REGION Network 5: создаем лог
   #_w1 := "data".executeCreate AND NOT #DL.stateMem;   // rising edge of "data".executeCreate
   #DL.stateMem := "data".executeCreate;
   #DataLogCreate_Instance(REQ := #_w1,   // DataLogCreate
                           RECORDS := 3000,
                           "NAME" := "data"."name",
                           ID := "data".logID,
                           DATA := "data".myData,
                           DONE => "data".crateDone,
                           BUSY => "data".createBusy,
                           ERROR => "data".createError,
                           STATUS => "data".createStatus);
END_REGION

REGION Network 6: если ошибка
   RUNG wire#powerrail
      Contact( "data".createError )
      Move(in := "data".createStatus, out1 => "data".createStatusMem)
   END_RUNG
   // the same network as SCL:
   IF "data".createError THEN "data".createStatusMem := "data".createStatus; END_IF;
END_REGION

REGION Network 7: создана сессия
   RUNG wire#powerrail
      Contact( "data".crateDone )
      S_Coil( "data".dlogCreated )
   END_RUNG
   // the same network as SCL:
   IF "data".crateDone THEN "data".dlogCreated := TRUE; END_IF;
END_REGION

REGION Network 8: запись значений в бд
   RUNG wire#powerrail
      P_Contact(operand := "logW".executeWrite, bit := #DL.stateMem_2)
      Move(in := "T3V3W3_DB".Statistic.Count, out1 => "data".myData.number)
      Move(in := "T3V3W3_DB".LocalVar.SP_loaded, out1 => "data".myData.weight)
   END_RUNG
   // the same network as SCL:
   #_w1 := "logW".executeWrite AND NOT #DL.stateMem_2;   // rising edge of "logW".executeWrite
   #DL.stateMem_2 := "logW".executeWrite;
   IF #_w1 THEN
       "data".myData.number := "T3V3W3_DB".Statistic.Count;
       "data".myData.weight := "T3V3W3_DB".LocalVar.SP_loaded;
   END_IF;
END_REGION

REGION Network 9: запись на флеш
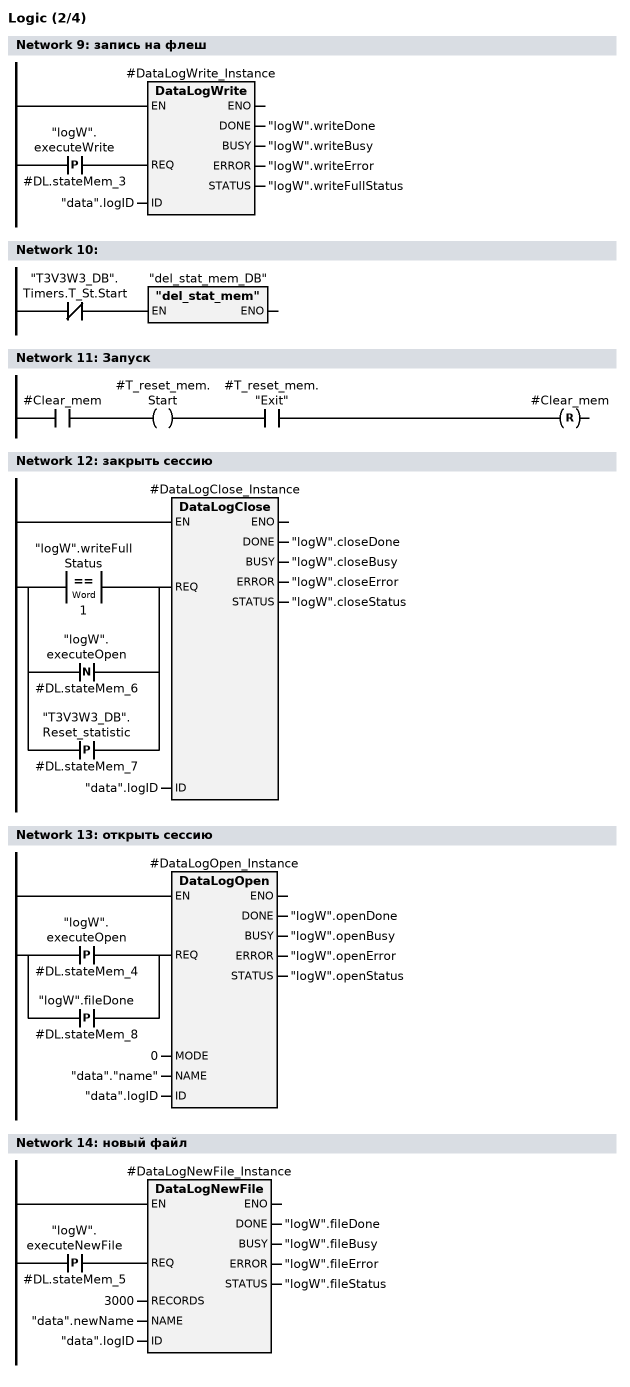
   #_w1 := "logW".executeWrite AND NOT #DL.stateMem_3;   // rising edge of "logW".executeWrite
   #DL.stateMem_3 := "logW".executeWrite;
   #DataLogWrite_Instance(REQ := #_w1,   // DataLogWrite
                          ID := "data".logID,
                          DONE => "logW".writeDone,
                          BUSY => "logW".writeBusy,
                          ERROR => "logW".writeError,
                          STATUS => "logW".writeFullStatus);
END_REGION

REGION Network 10
   RUNG wire#powerrail
      I_Contact( "T3V3W3_DB".Timers.T_St.Start )
      "del_stat_mem_DB"()
   END_RUNG
   // the same network as SCL:
   IF NOT "T3V3W3_DB".Timers.T_St.Start THEN
       "del_stat_mem_DB"();   // "del_stat_mem"
   END_IF;
END_REGION

REGION Network 11: Запуск
   RUNG wire#powerrail
      Contact( #Clear_mem )
      Coil( #T_reset_mem.Start )
      Contact( #T_reset_mem."Exit" )
      R_Coil( #Clear_mem )
   END_RUNG
   // the same network as SCL:
   #T_reset_mem.Start := #Clear_mem;
   IF #Clear_mem AND #T_reset_mem."Exit" THEN #Clear_mem := FALSE; END_IF;
END_REGION

REGION Network 12: закрыть сессию
   #_w1 := NOT "logW".executeOpen AND #DL.stateMem_6;   // falling edge of "logW".executeOpen
   #DL.stateMem_6 := "logW".executeOpen;
   #_w2 := "T3V3W3_DB".Reset_statistic AND NOT #DL.stateMem_7;   // rising edge of "T3V3W3_DB".Reset_statistic
   #DL.stateMem_7 := "T3V3W3_DB".Reset_statistic;
   #DataLogClose_Instance(REQ := ("logW".writeFullStatus = 1) OR #_w1 OR #_w2,   // DataLogClose
                          ID := "data".logID,
                          DONE => "logW".closeDone,
                          BUSY => "logW".closeBusy,
                          ERROR => "logW".closeError,
                          STATUS => "logW".closeStatus);
END_REGION

REGION Network 13: открыть сессию
   #_w1 := "logW".executeOpen AND NOT #DL.stateMem_4;   // rising edge of "logW".executeOpen
   #DL.stateMem_4 := "logW".executeOpen;
   #_w2 := "logW".fileDone AND NOT #DL.stateMem_8;   // rising edge of "logW".fileDone
   #DL.stateMem_8 := "logW".fileDone;
   #DataLogOpen_Instance(REQ := #_w1 OR #_w2,   // DataLogOpen
                         MODE := 0,
                         "NAME" := "data"."name",
                         ID := "data".logID,
                         DONE => "logW".openDone,
                         BUSY => "logW".openBusy,
                         ERROR => "logW".openError,
                         STATUS => "logW".openStatus);
END_REGION

REGION Network 14: новый файл
   #_w1 := "logW".executeNewFile AND NOT #DL.stateMem_5;   // rising edge of "logW".executeNewFile
   #DL.stateMem_5 := "logW".executeNewFile;
   #DataLogNewFile_Instance(REQ := #_w1,   // DataLogNewFile
                           RECORDS := 3000,
                           "NAME" := "data".newName,
                           ID := "data".logID,
                           DONE => "logW".fileDone,
                           BUSY => "logW".fileBusy,
                           ERROR => "logW".fileError,
                           STATUS => "logW".fileStatus);
END_REGION

REGION Network 16: Сброс команды на запись
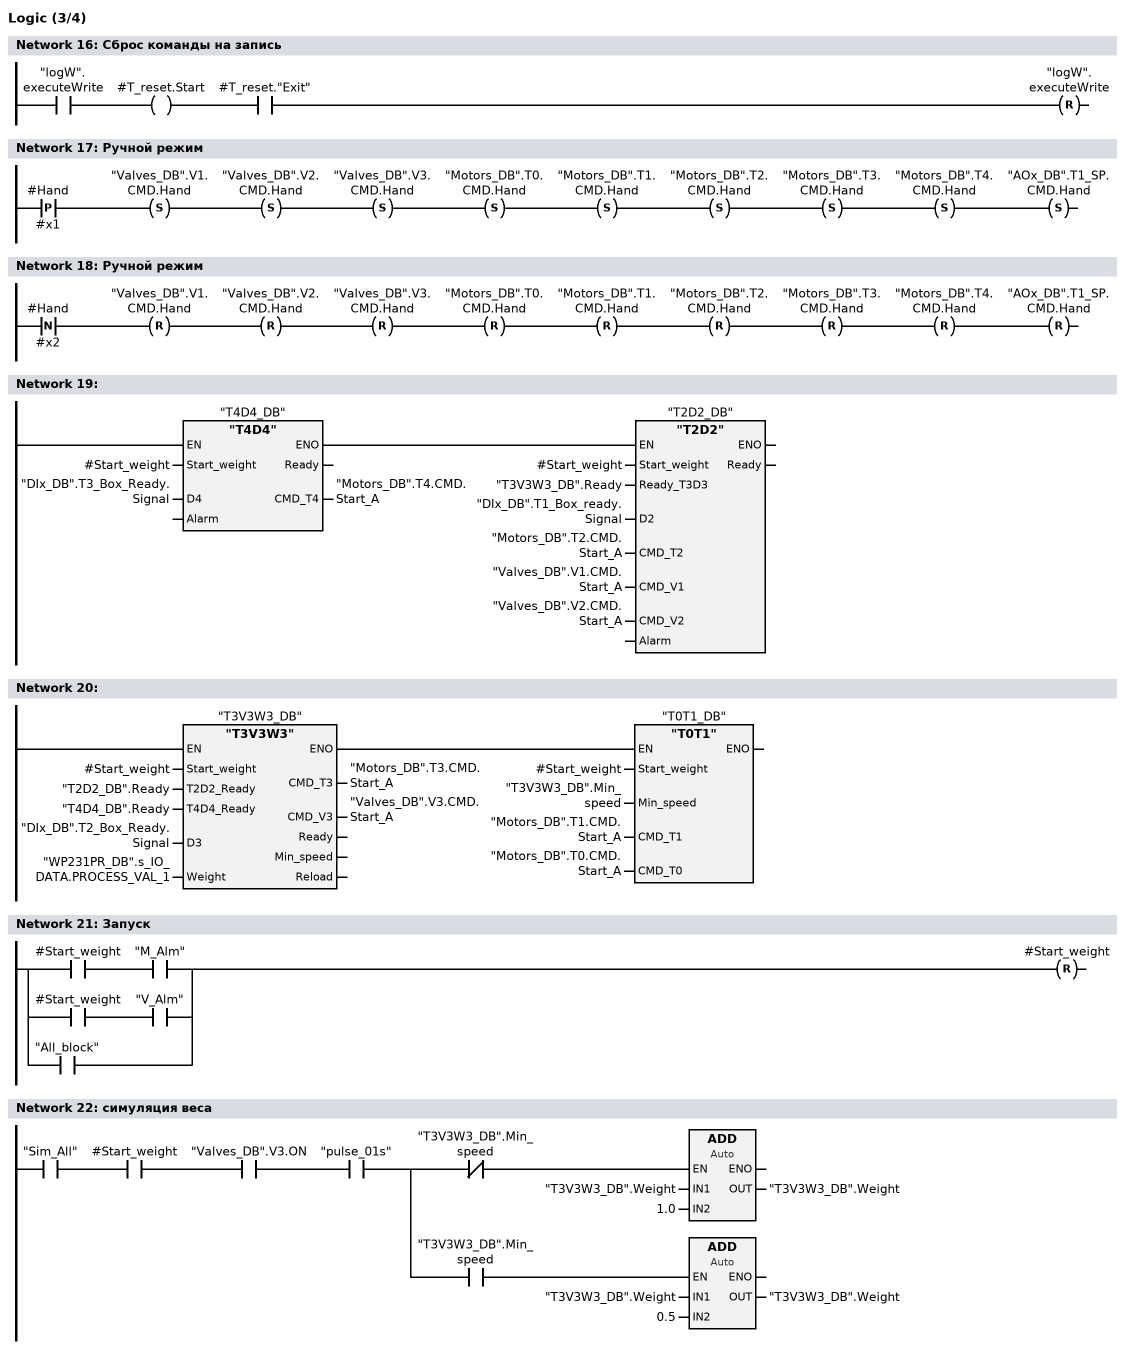
   RUNG wire#powerrail
      Contact( "logW".executeWrite )
      Coil( #T_reset.Start )
      Contact( #T_reset."Exit" )
      R_Coil( "logW".executeWrite )
   END_RUNG
   // the same network as SCL:
   #T_reset.Start := "logW".executeWrite;
   IF "logW".executeWrite AND #T_reset."Exit" THEN "logW".executeWrite := FALSE; END_IF;
END_REGION

REGION Network 17: Ручной режим
   RUNG wire#powerrail
      P_Contact(operand := #Hand, bit := #x1)
      S_Coil( "Valves_DB".V1.CMD.Hand )
      S_Coil( "Valves_DB".V2.CMD.Hand )
      S_Coil( "Valves_DB".V3.CMD.Hand )
      S_Coil( "Motors_DB".T0.CMD.Hand )
      S_Coil( "Motors_DB".T1.CMD.Hand )
      S_Coil( "Motors_DB".T2.CMD.Hand )
      S_Coil( "Motors_DB".T3.CMD.Hand )
      S_Coil( "Motors_DB".T4.CMD.Hand )
      S_Coil( "AOx_DB".T1_SP.CMD.Hand )
   END_RUNG
   // the same network as SCL:
   #_w1 := #Hand AND NOT #x1;   // rising edge of #Hand
   #x1 := #Hand;
   IF #_w1 THEN
       "Valves_DB".V1.CMD.Hand := TRUE;
       "Valves_DB".V2.CMD.Hand := TRUE;
       "Valves_DB".V3.CMD.Hand := TRUE;
       "Motors_DB".T0.CMD.Hand := TRUE;
       "Motors_DB".T1.CMD.Hand := TRUE;
       "Motors_DB".T2.CMD.Hand := TRUE;
       "Motors_DB".T3.CMD.Hand := TRUE;
       "Motors_DB".T4.CMD.Hand := TRUE;
       "AOx_DB".T1_SP.CMD.Hand := TRUE;
   END_IF;
END_REGION

REGION Network 18: Ручной режим
   RUNG wire#powerrail
      N_Contact(operand := #Hand, bit := #x2)
      R_Coil( "Valves_DB".V1.CMD.Hand )
      R_Coil( "Valves_DB".V2.CMD.Hand )
      R_Coil( "Valves_DB".V3.CMD.Hand )
      R_Coil( "Motors_DB".T0.CMD.Hand )
      R_Coil( "Motors_DB".T1.CMD.Hand )
      R_Coil( "Motors_DB".T2.CMD.Hand )
      R_Coil( "Motors_DB".T3.CMD.Hand )
      R_Coil( "Motors_DB".T4.CMD.Hand )
      R_Coil( "AOx_DB".T1_SP.CMD.Hand )
   END_RUNG
   // the same network as SCL:
   #_w1 := NOT #Hand AND #x2;   // falling edge of #Hand
   #x2 := #Hand;
   IF #_w1 THEN
       "Valves_DB".V1.CMD.Hand := FALSE;
       "Valves_DB".V2.CMD.Hand := FALSE;
       "Valves_DB".V3.CMD.Hand := FALSE;
       "Motors_DB".T0.CMD.Hand := FALSE;
       "Motors_DB".T1.CMD.Hand := FALSE;
       "Motors_DB".T2.CMD.Hand := FALSE;
       "Motors_DB".T3.CMD.Hand := FALSE;
       "Motors_DB".T4.CMD.Hand := FALSE;
       "AOx_DB".T1_SP.CMD.Hand := FALSE;
   END_IF;
END_REGION

REGION Network 19
   RUNG wire#powerrail
      "T4D4_DB"(Start_weight := #Start_weight, D4 := "DIx_DB".T3_Box_Ready.Signal, Alarm :=, Ready =>, CMD_T4 => "Motors_DB".T4.CMD.Start_A)
      "T2D2_DB"(Start_weight := #Start_weight, Ready_T3D3 := "T3V3W3_DB".Ready, D2 := "DIx_DB".T1_Box_ready.Signal, CMD_T2 := "Motors_DB".T2.CMD.Start_A, CMD_V1 := "Valves_DB".V1.CMD.Start_A, CMD_V2 := "Valves_DB".V2.CMD.Start_A, Alarm :=, Ready =>)
   END_RUNG
   // the same network as SCL:
   "T4D4_DB"(Start_weight := #Start_weight,   // "T4D4"
             D4 := "DIx_DB".T3_Box_Ready.Signal,
             CMD_T4 => "Motors_DB".T4.CMD.Start_A,
             ENO => #_w1);
   IF #_w1 THEN
       "T2D2_DB"(Start_weight := #Start_weight,   // "T2D2"
                 Ready_T3D3 := "T3V3W3_DB".Ready,
                 D2 := "DIx_DB".T1_Box_ready.Signal,
                 CMD_T2 := "Motors_DB".T2.CMD.Start_A,
                 CMD_V1 := "Valves_DB".V1.CMD.Start_A,
                 CMD_V2 := "Valves_DB".V2.CMD.Start_A);
   END_IF;
END_REGION

REGION Network 20
   RUNG wire#powerrail
      "T3V3W3_DB"(Start_weight := #Start_weight, T2D2_Ready := "T2D2_DB".Ready, T4D4_Ready := "T4D4_DB".Ready, D3 := "DIx_DB".T2_Box_Ready.Signal, Weight := "WP231PR_DB".s_IO_DATA.PROCESS_VAL_1, CMD_T3 => "Motors_DB".T3.CMD.Start_A, CMD_V3 => "Valves_DB".V3.CMD.Start_A, Ready =>, Min_speed =>, Reload =>)
      "T0T1_DB"(Start_weight := #Start_weight, Min_speed := "T3V3W3_DB".Min_speed, CMD_T1 := "Motors_DB".T1.CMD.Start_A, CMD_T0 := "Motors_DB".T0.CMD.Start_A)
   END_RUNG
   // the same network as SCL:
   "T3V3W3_DB"(Start_weight := #Start_weight,   // "T3V3W3"
               T2D2_Ready := "T2D2_DB".Ready,
               T4D4_Ready := "T4D4_DB".Ready,
               D3 := "DIx_DB".T2_Box_Ready.Signal,
               Weight := "WP231PR_DB".s_IO_DATA.PROCESS_VAL_1,
               CMD_T3 => "Motors_DB".T3.CMD.Start_A,
               CMD_V3 => "Valves_DB".V3.CMD.Start_A,
               ENO => #_w1);
   IF #_w1 THEN
       "T0T1_DB"(Start_weight := #Start_weight,   // "T0T1"
                 Min_speed := "T3V3W3_DB".Min_speed,
                 CMD_T1 := "Motors_DB".T1.CMD.Start_A,
                 CMD_T0 := "Motors_DB".T0.CMD.Start_A);
   END_IF;
END_REGION

REGION Network 21: Запуск
   RUNG wire#powerrail
      Contact( #Start_weight )
      Contact( "M_Alm" )
      wire#w1
      R_Coil( #Start_weight )
   END_RUNG
   RUNG wire#powerrail
      Contact( #Start_weight )
      Contact( "V_Alm" )
   END_RUNG wire#w1
   RUNG wire#powerrail
      Contact( "All_block" )
   END_RUNG wire#w1
   // the same network as SCL:
   IF (#Start_weight AND "M_Alm") OR (#Start_weight AND "V_Alm") OR "All_block" THEN
       #Start_weight := FALSE;
   END_IF;
END_REGION

REGION Network 22: симуляция веса
   RUNG wire#powerrail
      Contact( "Sim_All" )
      Contact( #Start_weight )
      Contact( "Valves_DB".V3.ON )
      Contact( "pulse_01s" )
      wire#w1
      I_Contact( "T3V3W3_DB".Min_speed )
      Add(in1 := "T3V3W3_DB".Weight, in2 := 1.0, out => "T3V3W3_DB".Weight)
   END_RUNG
   RUNG wire#w1
      Contact( "T3V3W3_DB".Min_speed )
      Add(in1 := "T3V3W3_DB".Weight, in2 := 0.5, out => "T3V3W3_DB".Weight)
   END_RUNG
   // the same network as SCL:
   #_w1 := "Sim_All" AND #Start_weight AND "Valves_DB".V3.ON AND "pulse_01s";
   IF #_w1 AND NOT "T3V3W3_DB".Min_speed THEN "T3V3W3_DB".Weight := "T3V3W3_DB".Weight + 1.0; END_IF;
   IF #_w1 AND "T3V3W3_DB".Min_speed THEN "T3V3W3_DB".Weight := "T3V3W3_DB".Weight + 0.5; END_IF;
END_REGION

REGION Network 23: инициализация таймера
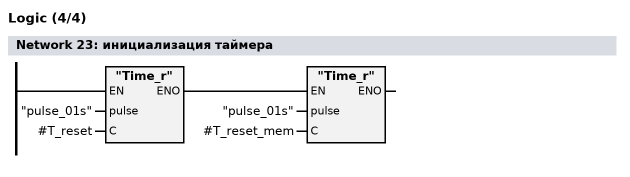
   RUNG wire#powerrail
      "Time_r"(pulse := "pulse_01s", C := #T_reset)
      "Time_r"(pulse := "pulse_01s", C := #T_reset_mem)
   END_RUNG
   // the same network as SCL:
   "Time_r"(pulse := "pulse_01s", C := #T_reset, ENO => #_w1);
   IF #_w1 THEN "Time_r"(pulse := "pulse_01s", C := #T_reset_mem); END_IF;
END_REGION
END_FUNCTION_BLOCK

FUNCTION_BLOCK "T3V3W3"   // FB10, LAD
{ S7_Optimized_Access := 'FALSE' }
VERSION : 0.1
   VAR_INPUT
      Start_weight : Bool;
      T2D2_Ready : Bool;
      T4D4_Ready : Bool;
      D3 : Bool;
      Weight : Real;
   END_VAR
   VAR_OUTPUT
      CMD_T3 : Bool;
      CMD_V3 : Bool;
      Ready : Bool;
      Min_speed : Bool;
      Reload : Bool;
   END_VAR
   VAR
      Reset_statistic_temp : Bool;
      Reset_statistic : Bool;
      Flag_record : Bool;
      Flag_reset : Bool;
      Reset_weight : Bool;
      Continue : Bool;
      Skip_box : Bool;
      No_box : Bool;
      x0 : Bool;
      x1 : Bool;
      Timers : Struct
         T_s7 : Struct
            SP : Real := 0.5;   // Уставка
            Now : Real;   // Текущий счёт
            One : Real := 0.1;   // Вес импульса
            Progress : Real;   // Прогресс выполнения
            "Exit" : Bool;   // Счёт завершён
            Start : Bool;   // Запуск
            Pause : Bool;   // Пауза
            Reset : Bool;   // Сброс счёта
            pos : Bool;   // Контроль фронта сигнала
         END_STRUCT;
         T_s15 : Struct
            SP : Real := 0.5;   // Уставка
            Now : Real;   // Текущий счёт
            One : Real := 0.1;   // Вес импульса
            Progress : Real;   // Прогресс выполнения
            "Exit" : Bool;   // Счёт завершён
            Start : Bool;   // Запуск
            Pause : Bool;   // Пауза
            Reset : Bool;   // Сброс счёта
            pos : Bool;   // Контроль фронта сигнала
         END_STRUCT;
         T_St : Struct
            SP : Real := 0.5;   // Уставка
            Now : Real;   // Текущий счёт
            One : Real := 0.1;   // Вес импульса
            Progress : Real;   // Прогресс выполнения
            "Exit" : Bool;   // Счёт завершён
            Start : Bool;   // Запуск
            Pause : Bool;   // Пауза
            Reset : Bool;   // Сброс счёта
            pos : Bool;   // Контроль фронта сигнала
         END_STRUCT;
      END_STRUCT;
      SetPoints : Struct
         SP : Real := 20.0;
         SP_fly : Real := 0.1;
         SP_ch_s : Real := 3.0;
         delta_add : Real := 0.2;
         delata_sub : Real := 0.1;
         count_reset : Int := 3000;
         count_warning : Int := 2500;
      END_STRUCT;
      LocalVar : Struct
         SP_load : Real;
         SP_loaded : Real;
         SP_max : Real;
         SP_min : Real;
         Sp_start : Real;
         Sp_ch_s_temp : Real;
         Temp_stat : Int;
         part_count : Int;
         len_str : Int;
         name_part : String := 'first';
         temp_id : DInt := 0;
      END_STRUCT;
      Statistic : Struct
         Count : Int;
         Weight : Real;
         Mid_weight : Real;
         Count_old : Int;
         Weight_old : Real;
         Mid_weight_old : Real;
         Count_no_ok : Int;
      END_STRUCT;
      "Step" : Int;
      flag : Int := 1;
      Alarm : Word;
      func_reset_Instance : "func_reset";
      part_names : Array[0..19] of String;
   END_VAR
   VAR_TEMP   // added for the SCL form of the ladder/FBD networks
      _w1 : Bool;
      _w2 : Bool;
      _w3 : Bool;
   END_VAR
BEGIN

REGION Network 1
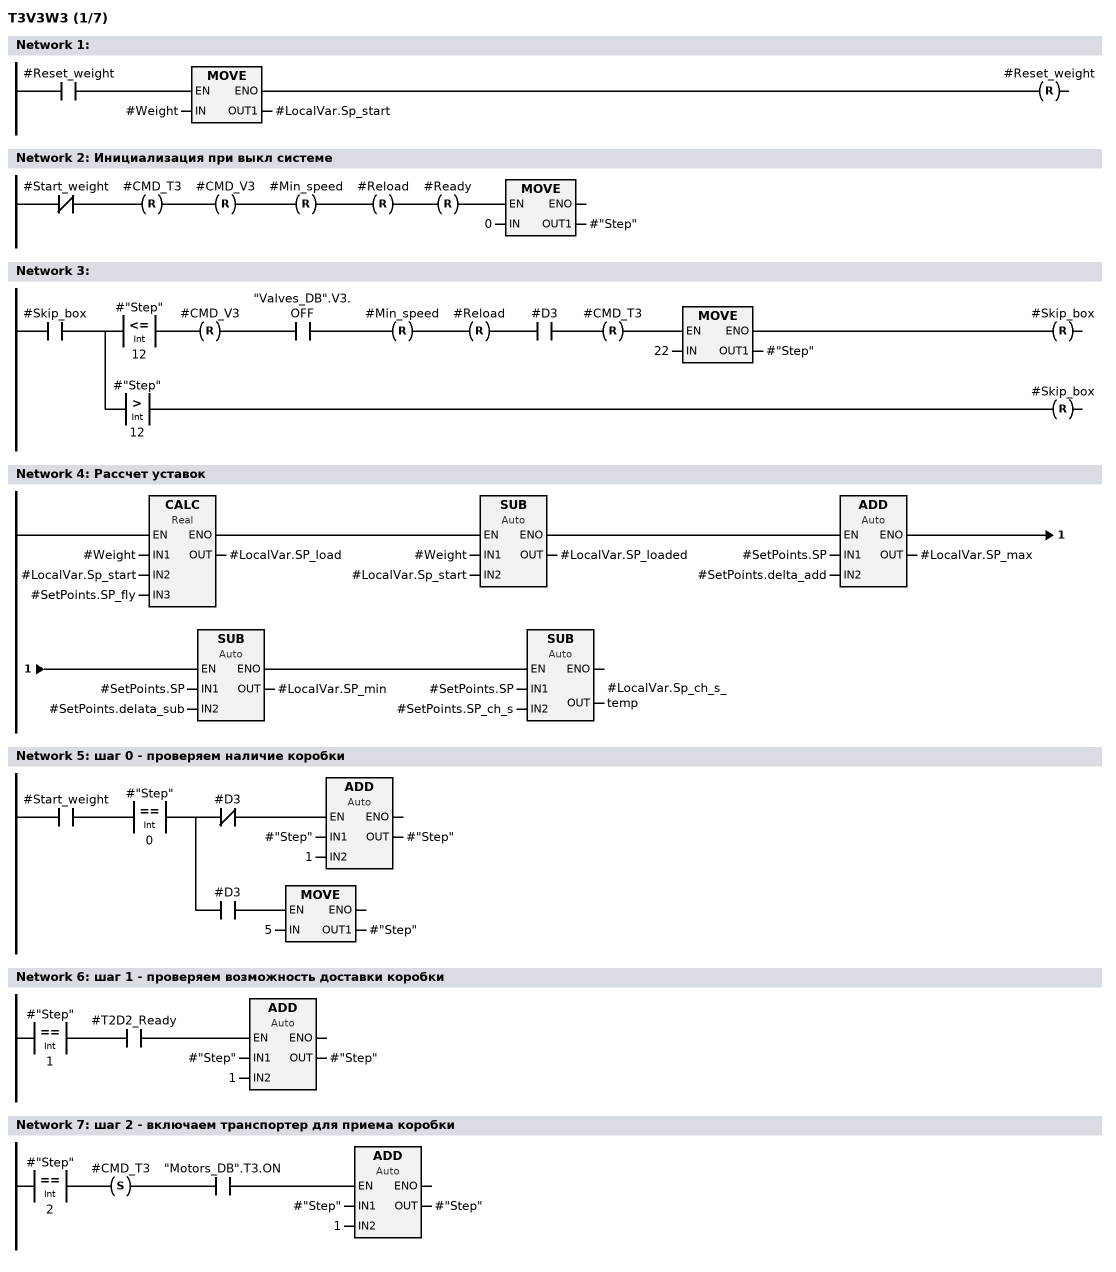
   RUNG wire#powerrail
      Contact( #Reset_weight )
      Move(in := #Weight, out1 => #LocalVar.Sp_start)
      R_Coil( #Reset_weight )
   END_RUNG
   // the same network as SCL:
   IF #Reset_weight THEN
       #LocalVar.Sp_start := #Weight;
       #Reset_weight := FALSE;
   END_IF;
END_REGION

REGION Network 2: Инициализация при выкл системе
   RUNG wire#powerrail
      I_Contact( #Start_weight )
      R_Coil( #CMD_T3 )
      R_Coil( #CMD_V3 )
      R_Coil( #Min_speed )
      R_Coil( #Reload )
      R_Coil( #Ready )
      Move(in := 0, out1 => #"Step")
   END_RUNG
   // the same network as SCL:
   IF NOT #Start_weight THEN
       #CMD_T3 := FALSE;
       #CMD_V3 := FALSE;
       #Min_speed := FALSE;
       #Reload := FALSE;
       #Ready := FALSE;
       #"Step" := 0;
   END_IF;
END_REGION

REGION Network 3
   RUNG wire#powerrail
      Contact( #Skip_box )
      wire#w1
      { S7_Templates := "SrcType := Int" } LE_Contact(in1 := #"Step", in2 := 12)
      R_Coil( #CMD_V3 )
      Contact( "Valves_DB".V3.OFF )
      R_Coil( #Min_speed )
      R_Coil( #Reload )
      Contact( #D3 )
      R_Coil( #CMD_T3 )
      Move(in := 22, out1 => #"Step")
      R_Coil( #Skip_box )
   END_RUNG
   RUNG wire#w1
      { S7_Templates := "SrcType := Int" } GT_Contact(in1 := #"Step", in2 := 12)
      R_Coil( #Skip_box )
   END_RUNG
   // the same network as SCL:
   #_w1 := #Skip_box AND (#"Step" <= 12);
   IF #_w1 THEN #CMD_V3 := FALSE; END_IF;
   #_w2 := #_w1 AND "Valves_DB".V3.OFF;
   IF #_w2 THEN
       #Min_speed := FALSE;
       #Reload := FALSE;
   END_IF;
   IF #_w2 AND #D3 THEN
       #CMD_T3 := FALSE;
       #"Step" := 22;
   END_IF;
   #_w3 := #Skip_box;
   IF #_w2 AND #D3 THEN #Skip_box := FALSE; END_IF;
   IF #_w3 AND (#"Step" > 12) THEN #Skip_box := FALSE; END_IF;
END_REGION

REGION Network 4: Рассчет уставок
   CALC(in1 := #Weight, in2 := #LocalVar.Sp_start, in3 := #SetPoints.SP_fly, out => #LocalVar.SP_load);
   #LocalVar.SP_loaded := #Weight - #LocalVar.Sp_start;
   #LocalVar.SP_max := #SetPoints.SP + #SetPoints.delta_add;
   #LocalVar.SP_min := #SetPoints.SP - #SetPoints.delata_sub;
   #LocalVar.Sp_ch_s_temp := #SetPoints.SP - #SetPoints.SP_ch_s;
END_REGION

REGION Network 5: шаг 0 - проверяем наличие коробки
   RUNG wire#powerrail
      Contact( #Start_weight )
      { S7_Templates := "SrcType := Int" } EQ_Contact(in1 := #"Step", in2 := 0)
      wire#w1
      I_Contact( #D3 )
      Add(in1 := #"Step", in2 := 1, out => #"Step")
   END_RUNG
   RUNG wire#w1
      Contact( #D3 )
      Move(in := 5, out1 => #"Step")
   END_RUNG
   // the same network as SCL:
   #_w1 := #Start_weight AND (#"Step" = 0);
   IF #_w1 AND NOT #D3 THEN #"Step" := #"Step" + 1; END_IF;
   IF #_w1 AND #D3 THEN #"Step" := 5; END_IF;
END_REGION

REGION Network 6: шаг 1 - проверяем возможность доставки коробки
   RUNG wire#powerrail
      { S7_Templates := "SrcType := Int" } EQ_Contact(in1 := #"Step", in2 := 1)
      Contact( #T2D2_Ready )
      Add(in1 := #"Step", in2 := 1, out => #"Step")
   END_RUNG
   // the same network as SCL:
   IF (#"Step" = 1) AND #T2D2_Ready THEN #"Step" := #"Step" + 1; END_IF;
END_REGION

REGION Network 7: шаг 2 - включаем транспортер для приема коробки
   RUNG wire#powerrail
      { S7_Templates := "SrcType := Int" } EQ_Contact(in1 := #"Step", in2 := 2)
      S_Coil( #CMD_T3 )
      Contact( "Motors_DB".T3.ON )
      Add(in1 := #"Step", in2 := 1, out => #"Step")
   END_RUNG
   // the same network as SCL:
   #_w1 := #"Step" = 2;
   IF #_w1 THEN #CMD_T3 := TRUE; END_IF;
   IF #_w1 AND "Motors_DB".T3.ON THEN #"Step" := #"Step" + 1; END_IF;
END_REGION

REGION Network 8: шаг 3 - устанавливаем готовность приема коробки
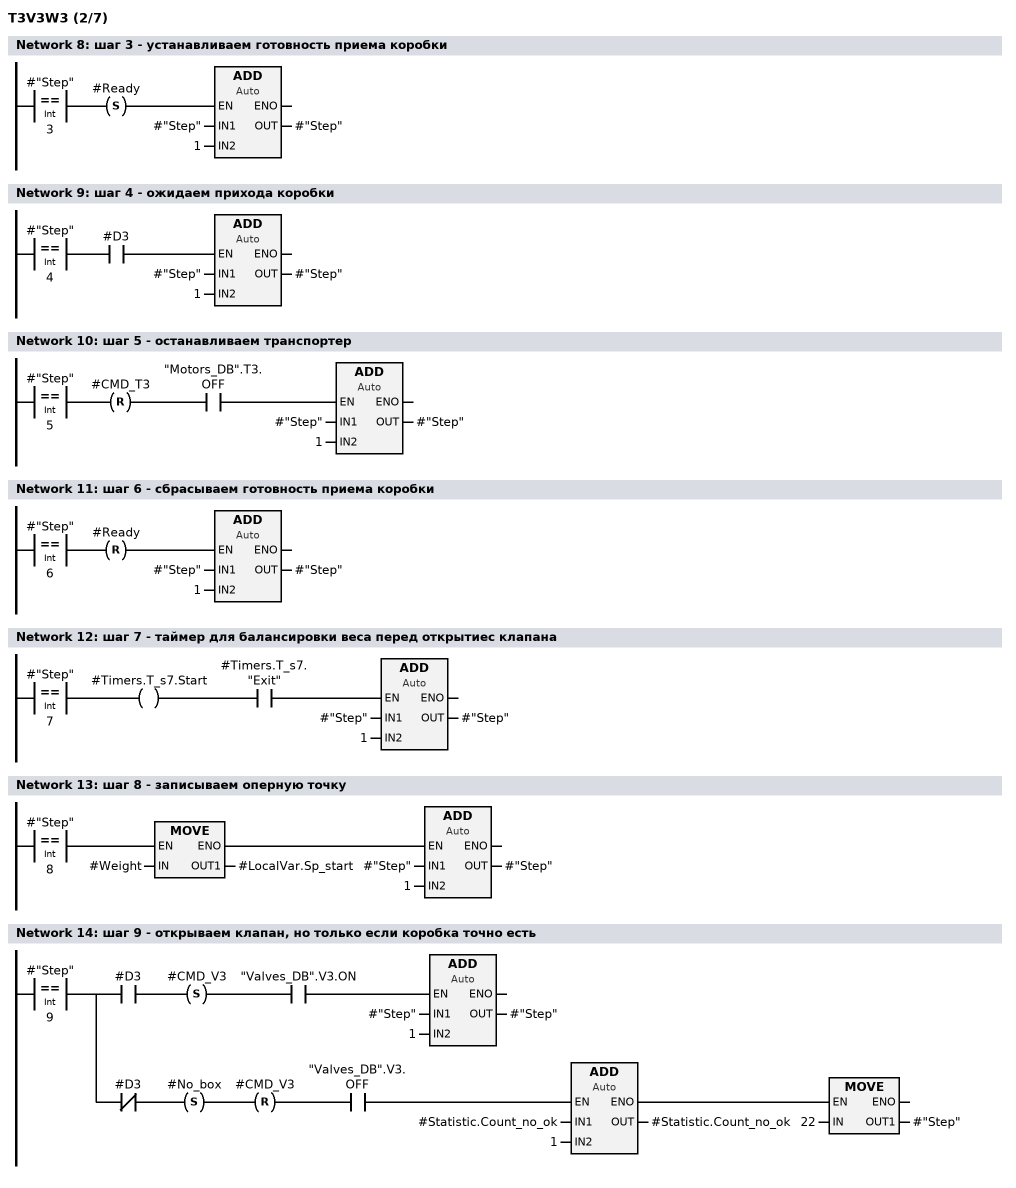
   RUNG wire#powerrail
      { S7_Templates := "SrcType := Int" } EQ_Contact(in1 := #"Step", in2 := 3)
      S_Coil( #Ready )
      Add(in1 := #"Step", in2 := 1, out => #"Step")
   END_RUNG
   // the same network as SCL:
   IF #"Step" = 3 THEN
       #Ready := TRUE;
       #"Step" := #"Step" + 1;
   END_IF;
END_REGION

REGION Network 9: шаг 4 - ожидаем прихода коробки
   RUNG wire#powerrail
      { S7_Templates := "SrcType := Int" } EQ_Contact(in1 := #"Step", in2 := 4)
      Contact( #D3 )
      Add(in1 := #"Step", in2 := 1, out => #"Step")
   END_RUNG
   // the same network as SCL:
   IF (#"Step" = 4) AND #D3 THEN #"Step" := #"Step" + 1; END_IF;
END_REGION

REGION Network 10: шаг 5 - останавливаем транспортер
   RUNG wire#powerrail
      { S7_Templates := "SrcType := Int" } EQ_Contact(in1 := #"Step", in2 := 5)
      R_Coil( #CMD_T3 )
      Contact( "Motors_DB".T3.OFF )
      Add(in1 := #"Step", in2 := 1, out => #"Step")
   END_RUNG
   // the same network as SCL:
   #_w1 := #"Step" = 5;
   IF #_w1 THEN #CMD_T3 := FALSE; END_IF;
   IF #_w1 AND "Motors_DB".T3.OFF THEN #"Step" := #"Step" + 1; END_IF;
END_REGION

REGION Network 11: шаг 6 - сбрасываем готовность приема коробки
   RUNG wire#powerrail
      { S7_Templates := "SrcType := Int" } EQ_Contact(in1 := #"Step", in2 := 6)
      R_Coil( #Ready )
      Add(in1 := #"Step", in2 := 1, out => #"Step")
   END_RUNG
   // the same network as SCL:
   IF #"Step" = 6 THEN
       #Ready := FALSE;
       #"Step" := #"Step" + 1;
   END_IF;
END_REGION

REGION Network 12: шаг 7 - таймер для балансировки веса перед открытиес клапана
   RUNG wire#powerrail
      { S7_Templates := "SrcType := Int" } EQ_Contact(in1 := #"Step", in2 := 7)
      Coil( #Timers.T_s7.Start )
      Contact( #Timers.T_s7."Exit" )
      Add(in1 := #"Step", in2 := 1, out => #"Step")
   END_RUNG
   // the same network as SCL:
   #Timers.T_s7.Start := #"Step" = 7;
   IF #Timers.T_s7.Start AND #Timers.T_s7."Exit" THEN #"Step" := #"Step" + 1; END_IF;
END_REGION

REGION Network 13: шаг 8 - записываем оперную точку
   RUNG wire#powerrail
      { S7_Templates := "SrcType := Int" } EQ_Contact(in1 := #"Step", in2 := 8)
      Move(in := #Weight, out1 => #LocalVar.Sp_start)
      Add(in1 := #"Step", in2 := 1, out => #"Step")
   END_RUNG
   // the same network as SCL:
   IF #"Step" = 8 THEN
       #LocalVar.Sp_start := #Weight;
       #"Step" := #"Step" + 1;
   END_IF;
END_REGION

REGION Network 14: шаг 9 - открываем клапан, но только если коробка точно есть
   RUNG wire#powerrail
      { S7_Templates := "SrcType := Int" } EQ_Contact(in1 := #"Step", in2 := 9)
      wire#w1
      Contact( #D3 )
      S_Coil( #CMD_V3 )
      Contact( "Valves_DB".V3.ON )
      Add(in1 := #"Step", in2 := 1, out => #"Step")
   END_RUNG
   RUNG wire#w1
      I_Contact( #D3 )
      S_Coil( #No_box )
      R_Coil( #CMD_V3 )
      Contact( "Valves_DB".V3.OFF )
      Add(in1 := #Statistic.Count_no_ok, in2 := 1, out => #Statistic.Count_no_ok)
      Move(in := 22, out1 => #"Step")
   END_RUNG
   // the same network as SCL:
   #_w1 := #"Step" = 9;
   #_w2 := #_w1 AND #D3;
   IF #_w2 THEN #CMD_V3 := TRUE; END_IF;
   IF #_w2 AND "Valves_DB".V3.ON THEN #"Step" := #"Step" + 1; END_IF;
   #_w3 := #_w1 AND NOT #D3;
   IF #_w3 THEN
       #No_box := TRUE;
       #CMD_V3 := FALSE;
   END_IF;
   IF #_w3 AND "Valves_DB".V3.OFF THEN
       #Statistic.Count_no_ok := #Statistic.Count_no_ok + 1;
       #"Step" := 22;
   END_IF;
END_REGION

REGION Network 15: шаг - 10 Ожидаем веса перехода на малую скорость
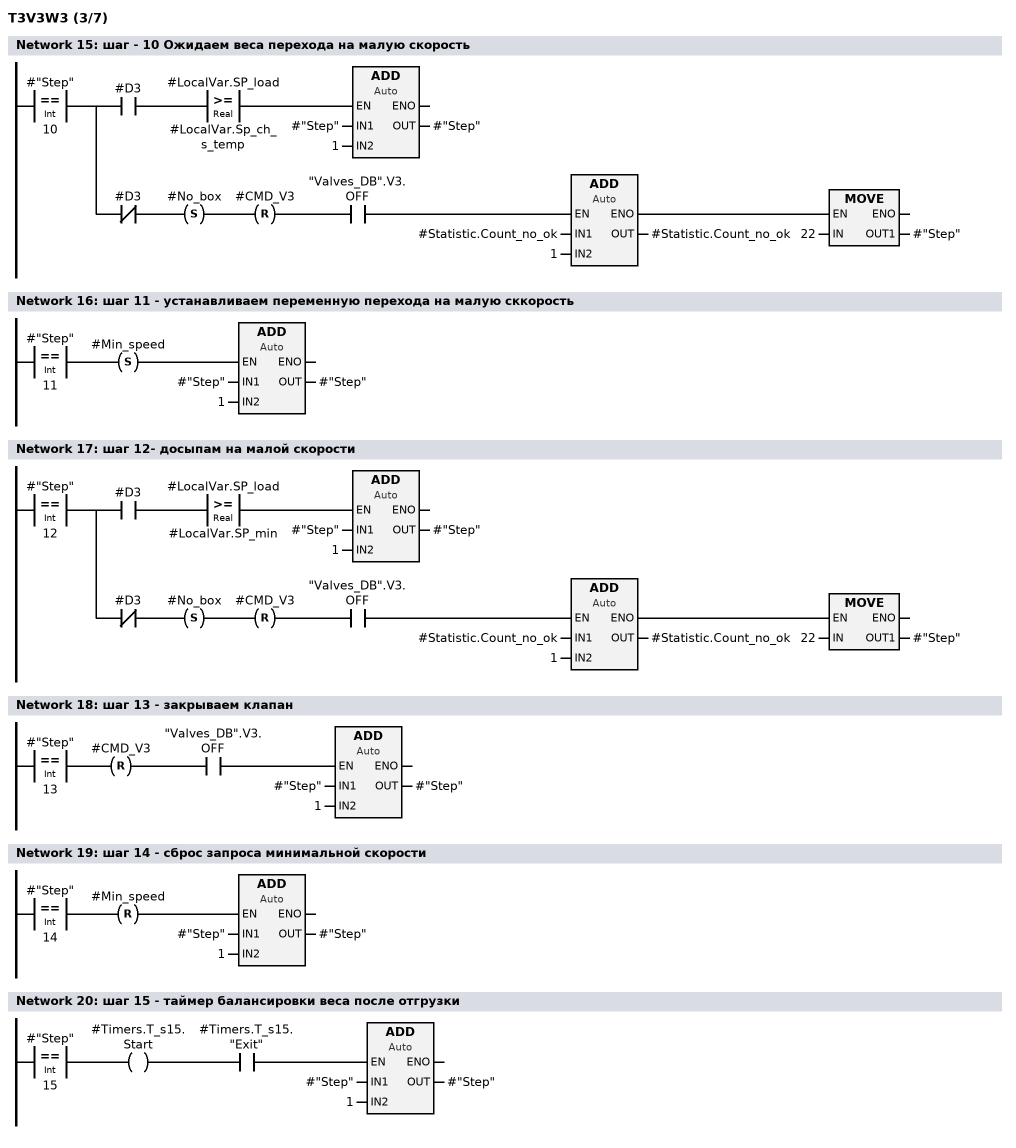
   RUNG wire#powerrail
      { S7_Templates := "SrcType := Int" } EQ_Contact(in1 := #"Step", in2 := 10)
      wire#w1
      Contact( #D3 )
      { S7_Templates := "SrcType := Real" } GE_Contact(in1 := #LocalVar.SP_load, in2 := #LocalVar.Sp_ch_s_temp)
      Add(in1 := #"Step", in2 := 1, out => #"Step")
   END_RUNG
   RUNG wire#w1
      I_Contact( #D3 )
      S_Coil( #No_box )
      R_Coil( #CMD_V3 )
      Contact( "Valves_DB".V3.OFF )
      Add(in1 := #Statistic.Count_no_ok, in2 := 1, out => #Statistic.Count_no_ok)
      Move(in := 22, out1 => #"Step")
   END_RUNG
   // the same network as SCL:
   #_w1 := #"Step" = 10;
   IF #_w1 AND #D3 AND (#LocalVar.SP_load >= #LocalVar.Sp_ch_s_temp) THEN #"Step" := #"Step" + 1; END_IF;
   #_w2 := #_w1 AND NOT #D3;
   IF #_w2 THEN
       #No_box := TRUE;
       #CMD_V3 := FALSE;
   END_IF;
   IF #_w2 AND "Valves_DB".V3.OFF THEN
       #Statistic.Count_no_ok := #Statistic.Count_no_ok + 1;
       #"Step" := 22;
   END_IF;
END_REGION

REGION Network 16: шаг 11 - устанавливаем переменную перехода на малую сккорость
   RUNG wire#powerrail
      { S7_Templates := "SrcType := Int" } EQ_Contact(in1 := #"Step", in2 := 11)
      S_Coil( #Min_speed )
      Add(in1 := #"Step", in2 := 1, out => #"Step")
   END_RUNG
   // the same network as SCL:
   IF #"Step" = 11 THEN
       #Min_speed := TRUE;
       #"Step" := #"Step" + 1;
   END_IF;
END_REGION

REGION Network 17: шаг 12- досыпам на малой скорости
   RUNG wire#powerrail
      { S7_Templates := "SrcType := Int" } EQ_Contact(in1 := #"Step", in2 := 12)
      wire#w1
      Contact( #D3 )
      { S7_Templates := "SrcType := Real" } GE_Contact(in1 := #LocalVar.SP_load, in2 := #LocalVar.SP_min)
      Add(in1 := #"Step", in2 := 1, out => #"Step")
   END_RUNG
   RUNG wire#w1
      I_Contact( #D3 )
      S_Coil( #No_box )
      R_Coil( #CMD_V3 )
      Contact( "Valves_DB".V3.OFF )
      Add(in1 := #Statistic.Count_no_ok, in2 := 1, out => #Statistic.Count_no_ok)
      Move(in := 22, out1 => #"Step")
   END_RUNG
   // the same network as SCL:
   #_w1 := #"Step" = 12;
   IF #_w1 AND #D3 AND (#LocalVar.SP_load >= #LocalVar.SP_min) THEN #"Step" := #"Step" + 1; END_IF;
   #_w2 := #_w1 AND NOT #D3;
   IF #_w2 THEN
       #No_box := TRUE;
       #CMD_V3 := FALSE;
   END_IF;
   IF #_w2 AND "Valves_DB".V3.OFF THEN
       #Statistic.Count_no_ok := #Statistic.Count_no_ok + 1;
       #"Step" := 22;
   END_IF;
END_REGION

REGION Network 18: шаг 13 - закрываем клапан
   RUNG wire#powerrail
      { S7_Templates := "SrcType := Int" } EQ_Contact(in1 := #"Step", in2 := 13)
      R_Coil( #CMD_V3 )
      Contact( "Valves_DB".V3.OFF )
      Add(in1 := #"Step", in2 := 1, out => #"Step")
   END_RUNG
   // the same network as SCL:
   #_w1 := #"Step" = 13;
   IF #_w1 THEN #CMD_V3 := FALSE; END_IF;
   IF #_w1 AND "Valves_DB".V3.OFF THEN #"Step" := #"Step" + 1; END_IF;
END_REGION

REGION Network 19: шаг 14 - сброс запроса минимальной скорости
   RUNG wire#powerrail
      { S7_Templates := "SrcType := Int" } EQ_Contact(in1 := #"Step", in2 := 14)
      R_Coil( #Min_speed )
      Add(in1 := #"Step", in2 := 1, out => #"Step")
   END_RUNG
   // the same network as SCL:
   IF #"Step" = 14 THEN
       #Min_speed := FALSE;
       #"Step" := #"Step" + 1;
   END_IF;
END_REGION

REGION Network 20: шаг 15 - таймер балансировки веса после отгрузки
   RUNG wire#powerrail
      { S7_Templates := "SrcType := Int" } EQ_Contact(in1 := #"Step", in2 := 15)
      Coil( #Timers.T_s15.Start )
      Contact( #Timers.T_s15."Exit" )
      Add(in1 := #"Step", in2 := 1, out => #"Step")
   END_RUNG
   // the same network as SCL:
   #Timers.T_s15.Start := #"Step" = 15;
   IF #Timers.T_s15.Start AND #Timers.T_s15."Exit" THEN #"Step" := #"Step" + 1; END_IF;
END_REGION

REGION Network 21: шаг 16 - сверка веса
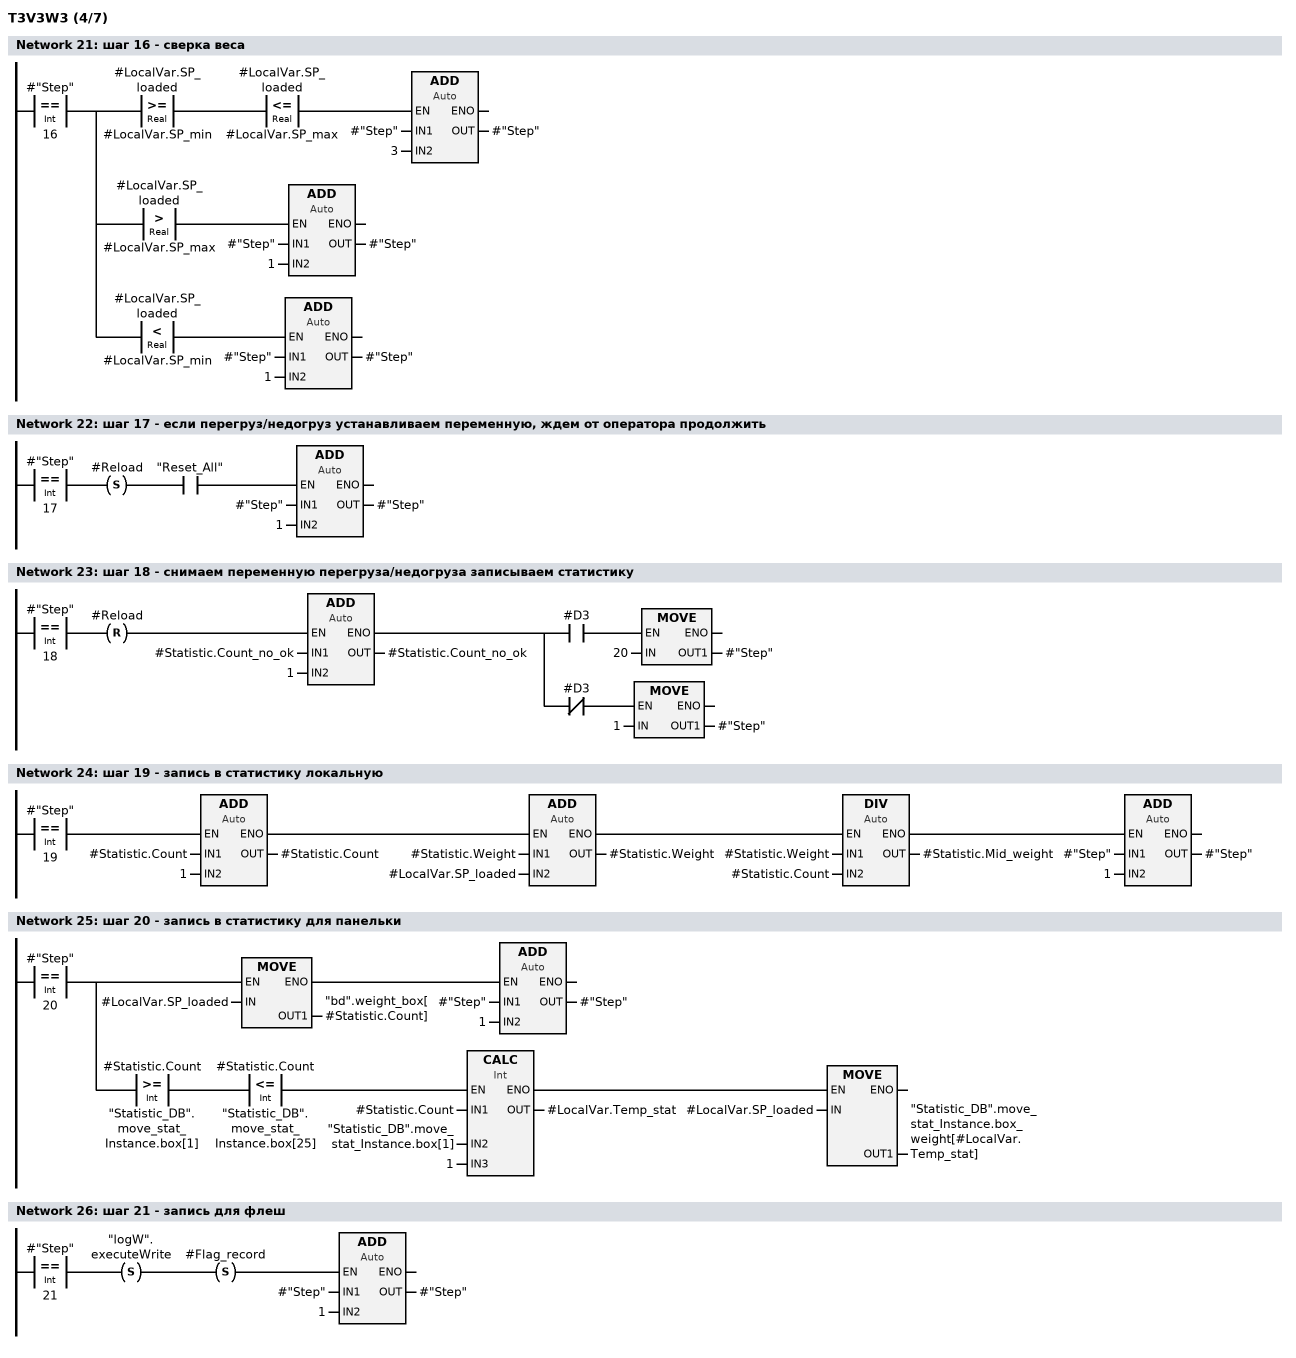
   RUNG wire#powerrail
      { S7_Templates := "SrcType := Int" } EQ_Contact(in1 := #"Step", in2 := 16)
      wire#w1
      { S7_Templates := "SrcType := Real" } GE_Contact(in1 := #LocalVar.SP_loaded, in2 := #LocalVar.SP_min)
      { S7_Templates := "SrcType := Real" } LE_Contact(in1 := #LocalVar.SP_loaded, in2 := #LocalVar.SP_max)
      Add(in1 := #"Step", in2 := 3, out => #"Step")
   END_RUNG
   RUNG wire#w1
      { S7_Templates := "SrcType := Real" } GT_Contact(in1 := #LocalVar.SP_loaded, in2 := #LocalVar.SP_max)
      Add(in1 := #"Step", in2 := 1, out => #"Step")
   END_RUNG
   RUNG wire#w1
      { S7_Templates := "SrcType := Real" } LT_Contact(in1 := #LocalVar.SP_loaded, in2 := #LocalVar.SP_min)
      Add(in1 := #"Step", in2 := 1, out => #"Step")
   END_RUNG
   // the same network as SCL:
   #_w1 := #"Step" = 16;
   IF #_w1 AND (#LocalVar.SP_loaded >= #LocalVar.SP_min) AND (#LocalVar.SP_loaded <= #LocalVar.SP_max) THEN
       #"Step" := #"Step" + 3;
   END_IF;
   IF #_w1 AND (#LocalVar.SP_loaded > #LocalVar.SP_max) THEN #"Step" := #"Step" + 1; END_IF;
   IF #_w1 AND (#LocalVar.SP_loaded < #LocalVar.SP_min) THEN #"Step" := #"Step" + 1; END_IF;
END_REGION

REGION Network 22: шаг 17 - если перегруз/недогруз устанавливаем переменную, ждем от оператора продолжить
   RUNG wire#powerrail
      { S7_Templates := "SrcType := Int" } EQ_Contact(in1 := #"Step", in2 := 17)
      S_Coil( #Reload )
      Contact( "Reset_All" )
      Add(in1 := #"Step", in2 := 1, out => #"Step")
   END_RUNG
   // the same network as SCL:
   #_w1 := #"Step" = 17;
   IF #_w1 THEN #Reload := TRUE; END_IF;
   IF #_w1 AND "Reset_All" THEN #"Step" := #"Step" + 1; END_IF;
END_REGION

REGION Network 23: шаг 18 - снимаем переменную перегруза/недогруза записываем статистику
   RUNG wire#powerrail
      { S7_Templates := "SrcType := Int" } EQ_Contact(in1 := #"Step", in2 := 18)
      R_Coil( #Reload )
      Add(in1 := #Statistic.Count_no_ok, in2 := 1, out => #Statistic.Count_no_ok)
      wire#w1
      Contact( #D3 )
      Move(in := 20, out1 => #"Step")
   END_RUNG
   RUNG wire#w1
      I_Contact( #D3 )
      Move(in := 1, out1 => #"Step")
   END_RUNG
   // the same network as SCL:
   #_w1 := #"Step" = 18;
   IF #_w1 THEN
       #Reload := FALSE;
       #Statistic.Count_no_ok := #Statistic.Count_no_ok + 1;
   END_IF;
   IF #_w1 AND #D3 THEN #"Step" := 20; END_IF;
   IF #_w1 AND NOT #D3 THEN #"Step" := 1; END_IF;
END_REGION

REGION Network 24: шаг 19 - запись в статистику локальную
   RUNG wire#powerrail
      { S7_Templates := "SrcType := Int" } EQ_Contact(in1 := #"Step", in2 := 19)
      Add(in1 := #Statistic.Count, in2 := 1, out => #Statistic.Count)
      Add(in1 := #Statistic.Weight, in2 := #LocalVar.SP_loaded, out => #Statistic.Weight)
      Div(in1 := #Statistic.Weight, in2 := #Statistic.Count, out => #Statistic.Mid_weight)
      Add(in1 := #"Step", in2 := 1, out => #"Step")
   END_RUNG
   // the same network as SCL:
   IF #"Step" = 19 THEN
       #Statistic.Count := #Statistic.Count + 1;
       #Statistic.Weight := #Statistic.Weight + #LocalVar.SP_loaded;
       #Statistic.Mid_weight := #Statistic.Weight / #Statistic.Count;
       #"Step" := #"Step" + 1;
   END_IF;
END_REGION

REGION Network 25: шаг 20 - запись в статистику для панельки
   #_w1 := #"Step" = 20;
   IF #_w1 THEN
       "bd".weight_box[#Statistic.Count] := #LocalVar.SP_loaded;
       #"Step" := #"Step" + 1;
   END_IF;
   #_w2 := #_w1 AND (#Statistic.Count >= "Statistic_DB".move_stat_Instance.box[1]) AND (#Statistic.Count <= "Statistic_DB".move_stat_Instance.box[25]);
   IF #_w2 THEN
       CALC(in1 := #Statistic.Count,
            in2 := "Statistic_DB".move_stat_Instance.box[1],
            in3 := 1,
            out => #LocalVar.Temp_stat);
       "Statistic_DB".move_stat_Instance.box_weight[#LocalVar.Temp_stat] := #LocalVar.SP_loaded;
   END_IF;
END_REGION

REGION Network 26: шаг 21 - запись для флеш
   RUNG wire#powerrail
      { S7_Templates := "SrcType := Int" } EQ_Contact(in1 := #"Step", in2 := 21)
      S_Coil( "logW".executeWrite )
      S_Coil( #Flag_record )
      Add(in1 := #"Step", in2 := 1, out => #"Step")
   END_RUNG
   // the same network as SCL:
   IF #"Step" = 21 THEN
       "logW".executeWrite := TRUE;
       #Flag_record := TRUE;
       #"Step" := #"Step" + 1;
   END_IF;
END_REGION

REGION Network 27: шаг 22 - проверяем готовность транспортером принять коробку
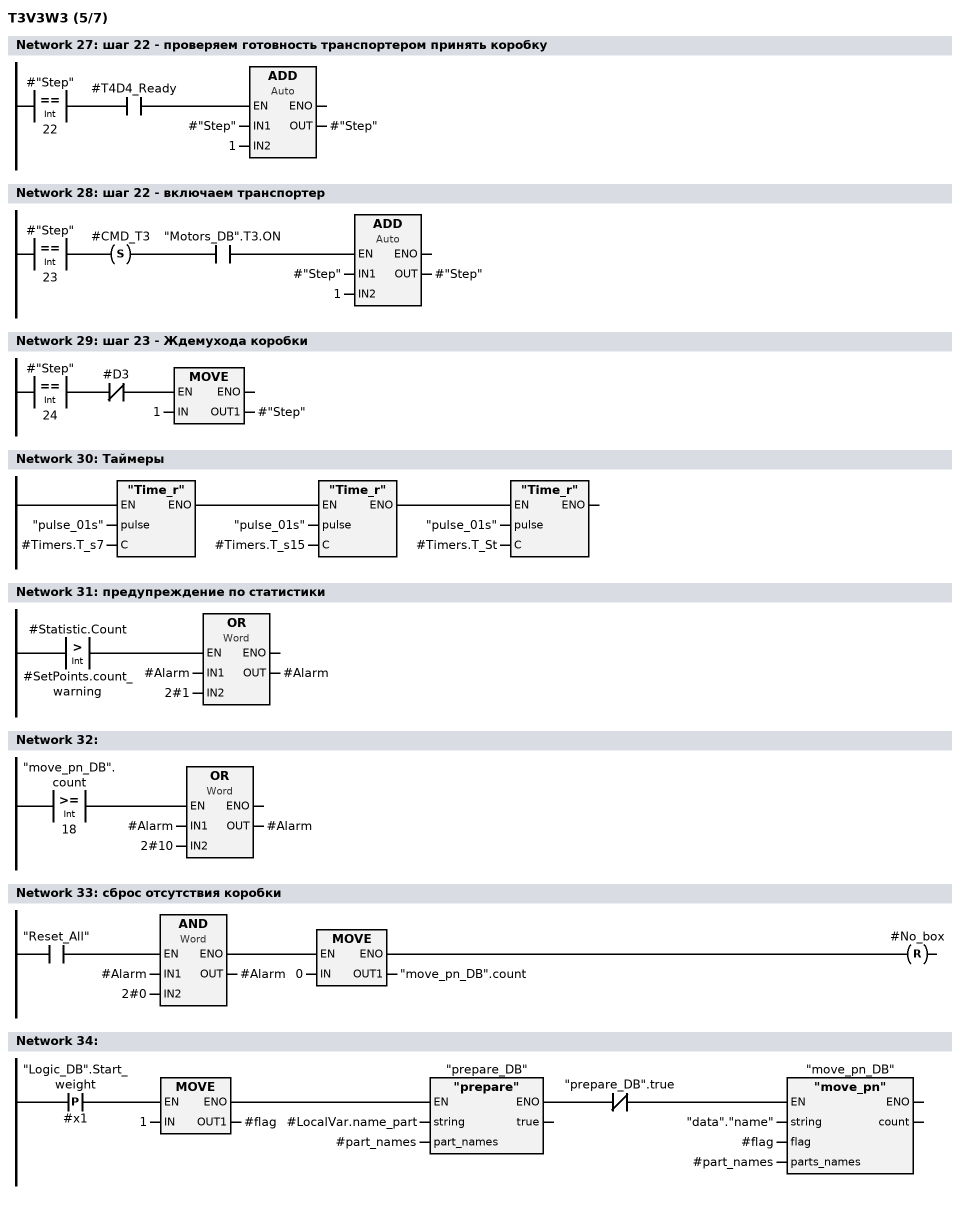
   RUNG wire#powerrail
      { S7_Templates := "SrcType := Int" } EQ_Contact(in1 := #"Step", in2 := 22)
      Contact( #T4D4_Ready )
      Add(in1 := #"Step", in2 := 1, out => #"Step")
   END_RUNG
   // the same network as SCL:
   IF (#"Step" = 22) AND #T4D4_Ready THEN #"Step" := #"Step" + 1; END_IF;
END_REGION

REGION Network 28: шаг 22 - включаем транспортер
   RUNG wire#powerrail
      { S7_Templates := "SrcType := Int" } EQ_Contact(in1 := #"Step", in2 := 23)
      S_Coil( #CMD_T3 )
      Contact( "Motors_DB".T3.ON )
      Add(in1 := #"Step", in2 := 1, out => #"Step")
   END_RUNG
   // the same network as SCL:
   #_w1 := #"Step" = 23;
   IF #_w1 THEN #CMD_T3 := TRUE; END_IF;
   IF #_w1 AND "Motors_DB".T3.ON THEN #"Step" := #"Step" + 1; END_IF;
END_REGION

REGION Network 29: шаг 23 - Ждемухода коробки
   RUNG wire#powerrail
      { S7_Templates := "SrcType := Int" } EQ_Contact(in1 := #"Step", in2 := 24)
      I_Contact( #D3 )
      Move(in := 1, out1 => #"Step")
   END_RUNG
   // the same network as SCL:
   IF (#"Step" = 24) AND NOT #D3 THEN #"Step" := 1; END_IF;
END_REGION

REGION Network 30: Таймеры
   RUNG wire#powerrail
      "Time_r"(pulse := "pulse_01s", C := #Timers.T_s7)
      "Time_r"(pulse := "pulse_01s", C := #Timers.T_s15)
      "Time_r"(pulse := "pulse_01s", C := #Timers.T_St)
   END_RUNG
   // the same network as SCL:
   "Time_r"(pulse := "pulse_01s", C := #Timers.T_s7, ENO => #_w1);
   "Time_r"(EN := #_w1, pulse := "pulse_01s", C := #Timers.T_s15, ENO => #_w2);
   IF #_w2 THEN "Time_r"(pulse := "pulse_01s", C := #Timers.T_St); END_IF;
END_REGION

REGION Network 31: предупреждение по статистики
   // no checked SCL form for this network; see the picture
END_REGION

REGION Network 32
   // no checked SCL form for this network; see the picture
END_REGION

REGION Network 33: сброс отсутствия коробки
   // no checked SCL form for this network; see the picture
END_REGION

REGION Network 34
   RUNG wire#powerrail
      P_Contact(operand := "Logic_DB".Start_weight, bit := #x1)
      Move(in := 1, out1 => #flag)
      "prepare_DB"("string" := #LocalVar.name_part, part_names := #part_names, true =>)
      I_Contact( "prepare_DB".true )
      "move_pn_DB"("string" := "data"."name", flag := #flag, parts_names := #part_names, count =>)
   END_RUNG
   // the same network as SCL:
   #_w1 := "Logic_DB".Start_weight AND NOT #x1;   // rising edge of "Logic_DB".Start_weight
   #x1 := "Logic_DB".Start_weight;
   IF #_w1 THEN #flag := 1; END_IF;
   "prepare_DB"(EN := #_w1, "string" := #LocalVar.name_part, part_names := #part_names, ENO => #_w2);   // "prepare"
   IF #_w2 AND NOT "prepare_DB".true THEN
       "move_pn_DB"("string" := "data"."name", flag := #flag, parts_names := #part_names);   // "move_pn"
   END_IF;
END_REGION

REGION Network 35
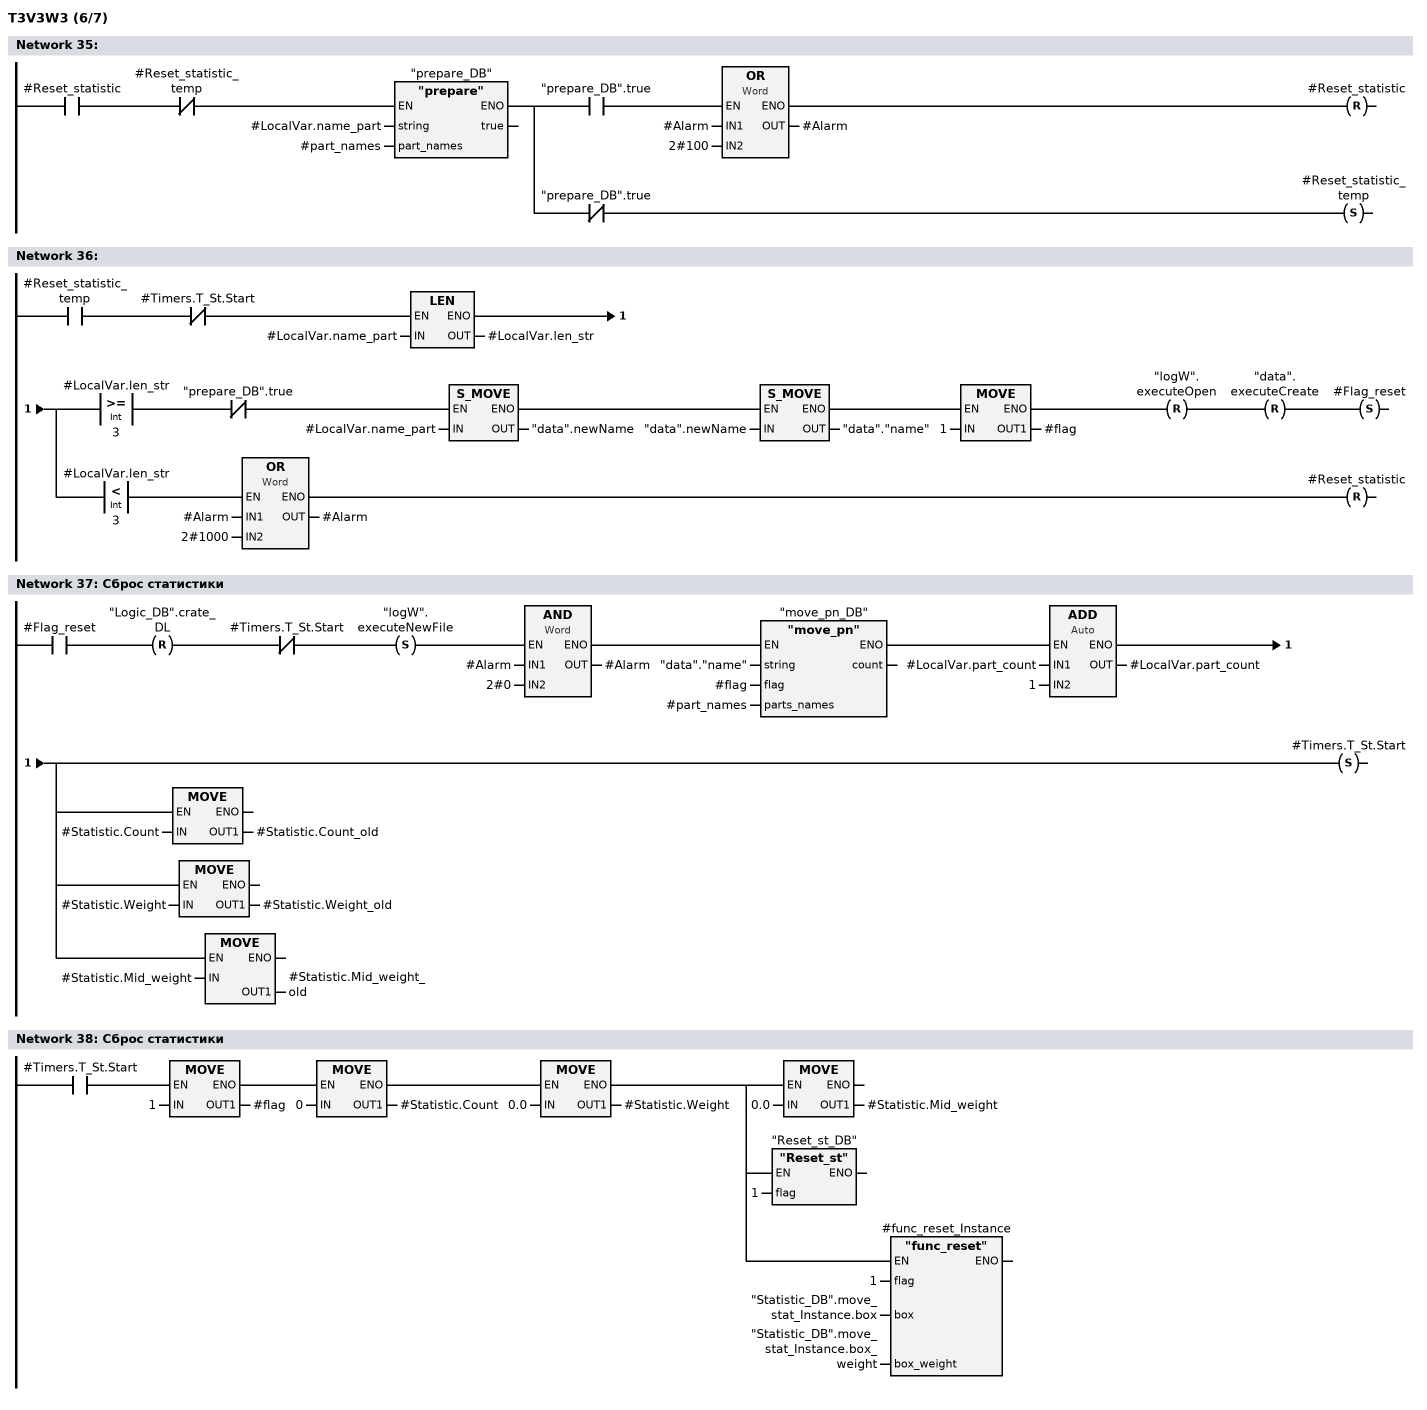
   // no checked SCL form for this network; see the picture
END_REGION

REGION Network 36
   // no checked SCL form for this network; see the picture
END_REGION

REGION Network 37: Сброс статистики
   // no checked SCL form for this network; see the picture
END_REGION

REGION Network 38: Сброс статистики
   RUNG wire#powerrail
      Contact( #Timers.T_St.Start )
      Move(in := 1, out1 => #flag)
      Move(in := 0, out1 => #Statistic.Count)
      Move(in := 0.0, out1 => #Statistic.Weight)
      wire#w1
      Move(in := 0.0, out1 => #Statistic.Mid_weight)
   END_RUNG
   RUNG wire#w1
      "Reset_st_DB"(flag := 1)
   END_RUNG
   RUNG wire#w1
      #func_reset_Instance(flag := 1, box := "Statistic_DB".move_stat_Instance.box, box_weight := "Statistic_DB".move_stat_Instance.box_weight)
   END_RUNG
   // the same network as SCL:
   IF #Timers.T_St.Start THEN
       #flag := 1;
       #Statistic.Count := 0;
       #Statistic.Weight := 0.0;
       #Statistic.Mid_weight := 0.0;
       "Reset_st_DB"(flag := 1);   // "Reset_st"
       #func_reset_Instance(flag := 1,   // "func_reset"
                            box := "Statistic_DB".move_stat_Instance.box,
                            box_weight := "Statistic_DB".move_stat_Instance.box_weight);
   END_IF;
END_REGION

REGION Network 39: Сброс статистики
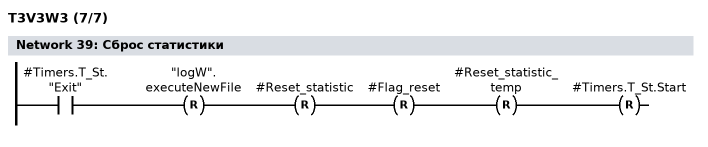
   RUNG wire#powerrail
      Contact( #Timers.T_St."Exit" )
      R_Coil( "logW".executeNewFile )
      R_Coil( #Reset_statistic )
      R_Coil( #Flag_reset )
      R_Coil( #Reset_statistic_temp )
      R_Coil( #Timers.T_St.Start )
   END_RUNG
   // the same network as SCL:
   IF #Timers.T_St."Exit" THEN
       "logW".executeNewFile := FALSE;
       #Reset_statistic := FALSE;
       #Flag_reset := FALSE;
       #Reset_statistic_temp := FALSE;
       #Timers.T_St.Start := FALSE;
   END_IF;
END_REGION
END_FUNCTION_BLOCK

FUNCTION_BLOCK "T2D2"   // FB11, LAD
{ S7_Optimized_Access := 'FALSE' }
VERSION : 0.1
   VAR_INPUT
      Start_weight : Bool;
      Ready_T3D3 : Bool;
      D2 : Bool;
   END_VAR
   VAR_OUTPUT
      Ready : Bool;
   END_VAR
   VAR_IN_OUT
      CMD_T2 : Bool;
      CMD_V1 : Bool;
      CMD_V2 : Bool;
      Alarm : Bool;
   END_VAR
   VAR
      "Step" : Int;
   END_VAR
BEGIN

REGION Network 1: Управление транспортером 2, вкл если открыт один из клапанов
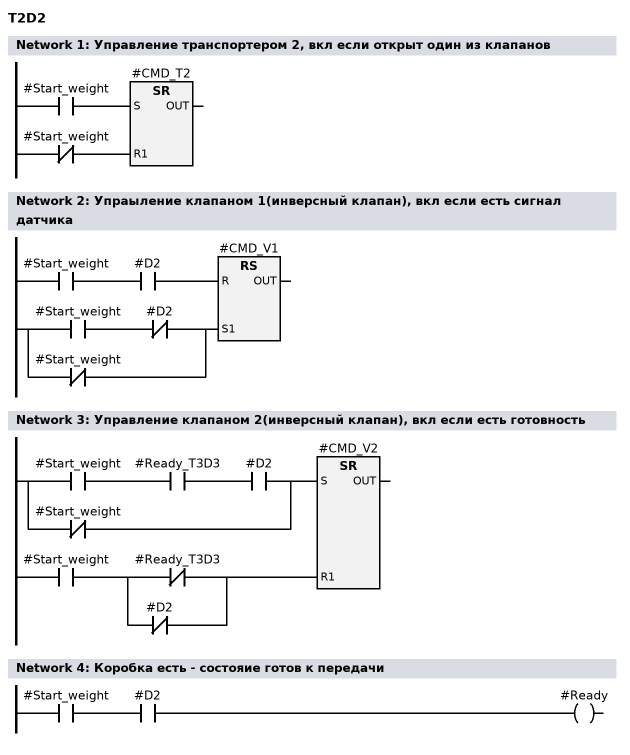
   RUNG wire#powerrail
      Contact( #Start_weight )
      S_SR(operand := #CMD_T2, r1 := wire#w1)
   END_RUNG
   RUNG wire#powerrail
      I_Contact( #Start_weight )
   END_RUNG wire#w1
   // the same network as SCL:
   IF #Start_weight THEN
       #CMD_T2 := TRUE;   // SR flip-flop
   END_IF;
   IF NOT #Start_weight THEN #CMD_T2 := FALSE; END_IF;
END_REGION

REGION Network 2: Упраыление клапаном 1(инверсный клапан), вкл если есть сигнал датчика
   RUNG wire#powerrail
      Contact( #Start_weight )
      Contact( #D2 )
      S_RS(operand := #CMD_V1, s1 := wire#w1)
   END_RUNG
   RUNG wire#powerrail
      Contact( #Start_weight )
      I_Contact( #D2 )
   END_RUNG wire#w1
   RUNG wire#powerrail
      I_Contact( #Start_weight )
   END_RUNG wire#w1
   // the same network as SCL:
   IF #Start_weight AND #D2 THEN
       #CMD_V1 := FALSE;   // RS flip-flop
   END_IF;
   IF (#Start_weight AND NOT #D2) OR NOT #Start_weight THEN #CMD_V1 := TRUE; END_IF;
END_REGION

REGION Network 3: Управление клапаном 2(инверсный клапан), вкл если есть готовность
   RUNG wire#powerrail
      Contact( #Start_weight )
      Contact( #Ready_T3D3 )
      Contact( #D2 )
      wire#w1
      S_SR(operand := #CMD_V2, r1 := wire#w3)
   END_RUNG
   RUNG wire#powerrail
      I_Contact( #Start_weight )
   END_RUNG wire#w1
   RUNG wire#powerrail
      Contact( #Start_weight )
      wire#w2
      I_Contact( #Ready_T3D3 )
   END_RUNG wire#w3
   RUNG wire#w2
      I_Contact( #D2 )
   END_RUNG wire#w3
   // the same network as SCL:
   IF (#Start_weight AND #Ready_T3D3 AND #D2) OR NOT #Start_weight THEN
       #CMD_V2 := TRUE;   // SR flip-flop
   END_IF;
   IF #Start_weight AND (NOT #Ready_T3D3 OR NOT #D2) THEN #CMD_V2 := FALSE; END_IF;
END_REGION

REGION Network 4: Коробка есть - состояие готов к передачи
   RUNG wire#powerrail
      Contact( #Start_weight )
      Contact( #D2 )
      Coil( #Ready )
   END_RUNG
   // the same network as SCL:
   #Ready := #Start_weight AND #D2;
END_REGION
END_FUNCTION_BLOCK

FUNCTION_BLOCK "T0T1"   // FB12, LAD
{ S7_Optimized_Access := 'FALSE' }
VERSION : 0.1
   VAR_INPUT
      Start_weight : Bool;
      Min_speed : Bool;
   END_VAR
   VAR_IN_OUT
      CMD_T1 : Bool;
      CMD_T0 : Bool;
   END_VAR
   VAR
      SP_min : Real := 30.0;
      SP_max : Real := 60.0;
   END_VAR
   VAR_TEMP   // added for the SCL form of the ladder/FBD networks
      _w1 : Bool;
   END_VAR
BEGIN

REGION Network 1
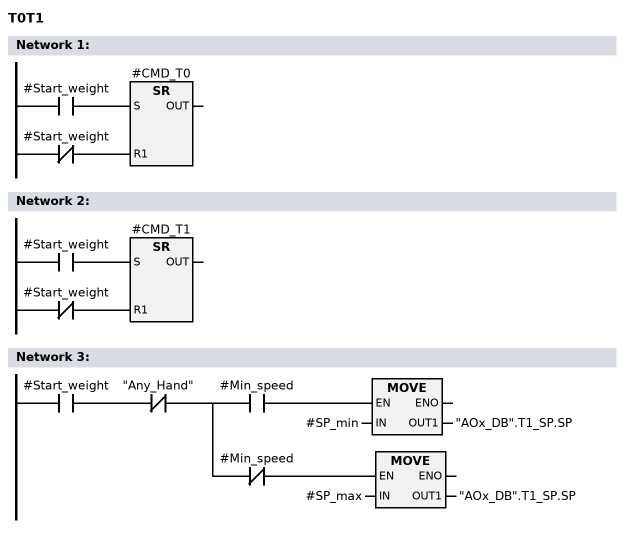
   RUNG wire#powerrail
      Contact( #Start_weight )
      S_SR(operand := #CMD_T0, r1 := wire#w1)
   END_RUNG
   RUNG wire#powerrail
      I_Contact( #Start_weight )
   END_RUNG wire#w1
   // the same network as SCL:
   IF #Start_weight THEN
       #CMD_T0 := TRUE;   // SR flip-flop
   END_IF;
   IF NOT #Start_weight THEN #CMD_T0 := FALSE; END_IF;
END_REGION

REGION Network 2
   RUNG wire#powerrail
      Contact( #Start_weight )
      S_SR(operand := #CMD_T1, r1 := wire#w1)
   END_RUNG
   RUNG wire#powerrail
      I_Contact( #Start_weight )
   END_RUNG wire#w1
   // the same network as SCL:
   IF #Start_weight THEN
       #CMD_T1 := TRUE;   // SR flip-flop
   END_IF;
   IF NOT #Start_weight THEN #CMD_T1 := FALSE; END_IF;
END_REGION

REGION Network 3
   RUNG wire#powerrail
      Contact( #Start_weight )
      I_Contact( "Any_Hand" )
      wire#w1
      Contact( #Min_speed )
      Move(in := #SP_min, out1 => "AOx_DB".T1_SP.SP)
   END_RUNG
   RUNG wire#w1
      I_Contact( #Min_speed )
      Move(in := #SP_max, out1 => "AOx_DB".T1_SP.SP)
   END_RUNG
   // the same network as SCL:
   #_w1 := #Start_weight AND NOT "Any_Hand";
   IF #_w1 AND #Min_speed THEN "AOx_DB".T1_SP.SP := #SP_min; END_IF;
   IF #_w1 AND NOT #Min_speed THEN "AOx_DB".T1_SP.SP := #SP_max; END_IF;
END_REGION
END_FUNCTION_BLOCK

FUNCTION_BLOCK "del_stat_mem"   // FB19, LAD
{ S7_Optimized_Access := 'FALSE' }
VERSION : 0.1
   VAR
      x0 : Bool;
      del_1 : Bool;
      del : Bool;
      count : Int;
      number : Int;
      flag : Int := 1;
      nul_str : String;
      DataLogDelete_Instance_1 : DataLogDelete;
      recombine_Instance : "move_pn";
      T_del : Struct
         SP : Real := 1.5;   // Уставка
         Now : Real;   // Текущий счёт
         One : Real := 0.1;   // Вес импульса
         Progress : Real;   // Прогресс выполнения
         "Exit" : Bool;   // Счёт завершён
         Start : Bool;   // Запуск
         Pause : Bool;   // Пауза
         Reset : Bool;   // Сброс счёта
         pos : Bool;   // Контроль фронта сигнала
      END_STRUCT;
      Alarm : Word;
   END_VAR
   VAR_TEMP   // added for the SCL form of the ladder/FBD networks
      _w1 : Bool;
      _w2 : Bool;
      _w3 : Bool;
      _w4 : Bool;
   END_VAR
BEGIN

REGION Network 1
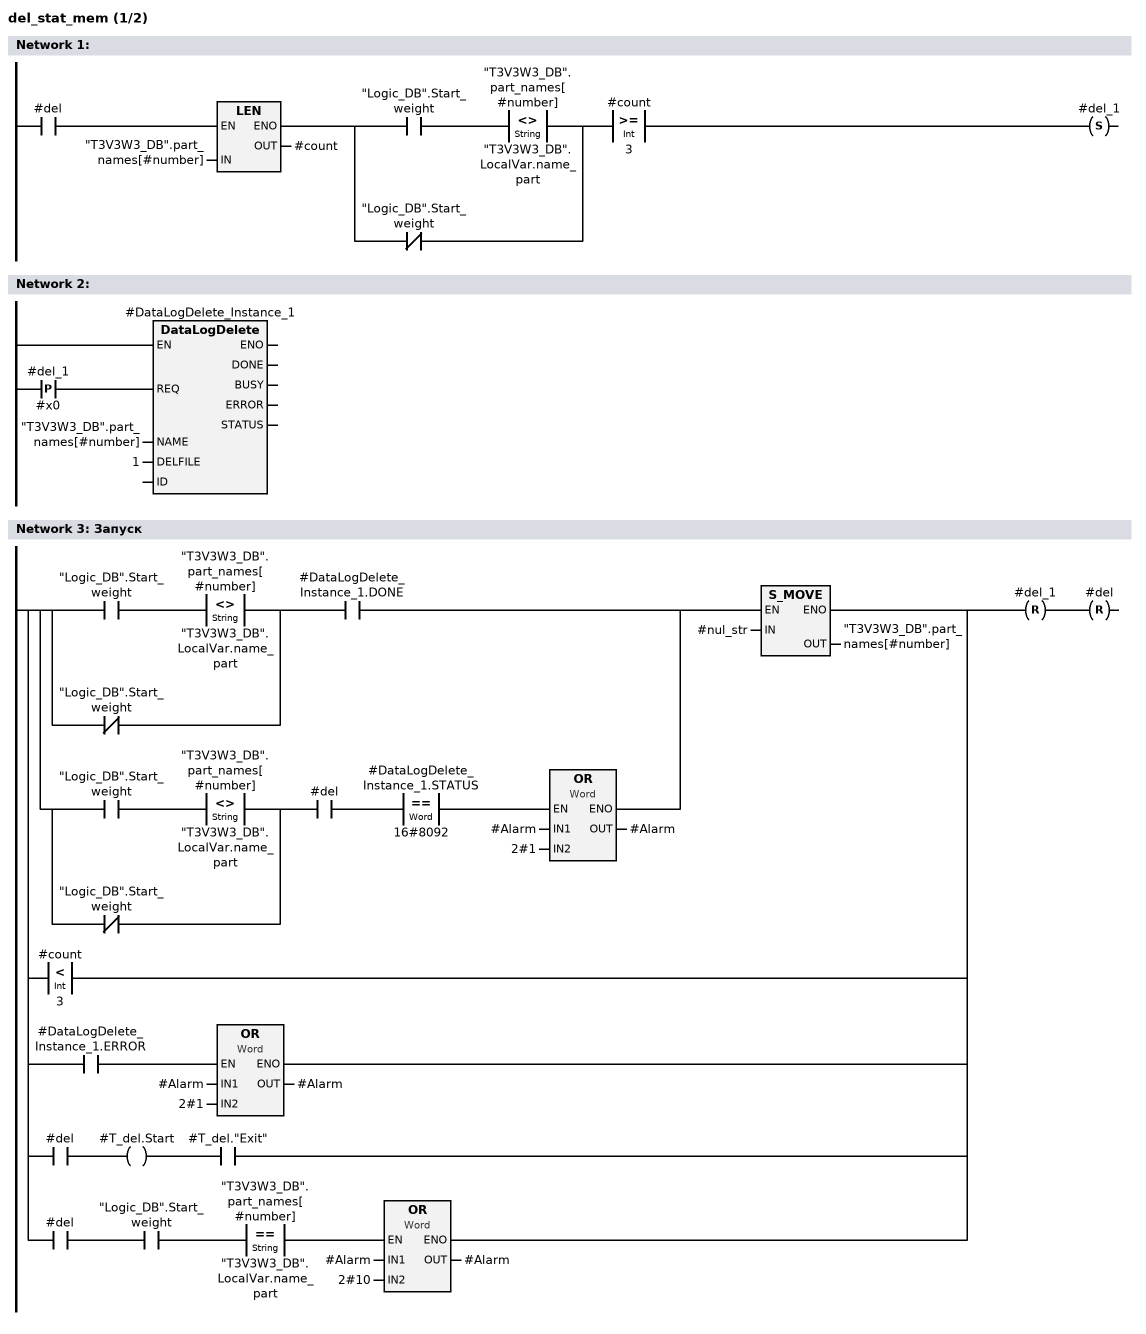
   IF #del THEN #count := LEN(IN := "T3V3W3_DB".part_names[#number]); END_IF;
   IF #del AND (("Logic_DB".Start_weight AND ("T3V3W3_DB".part_names[#number] <> "T3V3W3_DB".LocalVar.name_part)) OR NOT "Logic_DB".Start_weight) AND (#count >= 3) THEN
       #del_1 := TRUE;
   END_IF;
END_REGION

REGION Network 2
   #_w1 := #del_1 AND NOT #x0;   // rising edge of #del_1
   #x0 := #del_1;
   #DataLogDelete_Instance_1(REQ := #_w1, "NAME" := "T3V3W3_DB".part_names[#number], DelFile := 1);   // DataLogDelete
END_REGION

REGION Network 3: Запуск
   // no checked SCL form for this network; see the picture
END_REGION

REGION Network 4
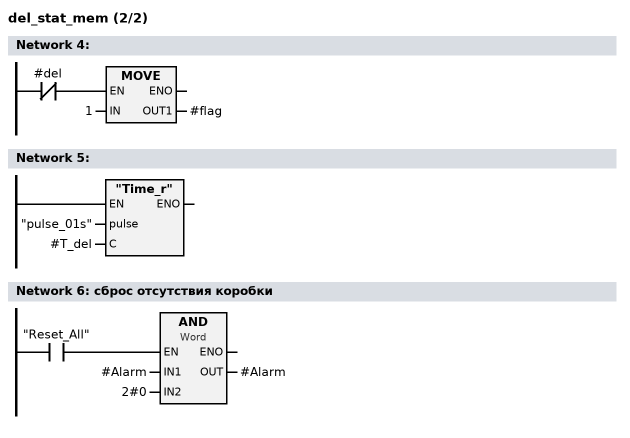
   RUNG wire#powerrail
      I_Contact( #del )
      Move(in := 1, out1 => #flag)
   END_RUNG
   // the same network as SCL:
   IF NOT #del THEN #flag := 1; END_IF;
END_REGION

REGION Network 5
   RUNG wire#powerrail
      "Time_r"(pulse := "pulse_01s", C := #T_del)
   END_RUNG
   // the same network as SCL:
   "Time_r"(pulse := "pulse_01s", C := #T_del);
END_REGION

REGION Network 6: сброс отсутствия коробки
   // no checked SCL form for this network; see the picture
END_REGION
END_FUNCTION_BLOCK

FUNCTION_BLOCK "move_pn"   // FB20, SCL
{ S7_Optimized_Access := 'FALSE' }
VERSION : 0.1
   VAR_INPUT
      "string" : String;
   END_VAR
   VAR_OUTPUT
      count : Int;
   END_VAR
   VAR_IN_OUT
      flag : Int;
      parts_names : Array[0..19] of String;
   END_VAR
   VAR
      i : Int;
   END_VAR
BEGIN
   IF #flag = 1 THEN
       #count := 0;
       FOR #i := 0 TO 19 DO
           IF LEN(#parts_names[#i]) < 3 AND #flag = 1 THEN
               #parts_names[#i] := #"string";
               #flag := 0;
           END_IF;
           IF LEN(#parts_names[#i]) >= 3 AND #flag = 1 THEN
               #count := #count + 1;
           END_IF;
       END_FOR;
   END_IF;
END_FUNCTION_BLOCK

FUNCTION_BLOCK "prepare"   // FB21, LAD
{ S7_Optimized_Access := 'TRUE' }
VERSION : 0.1
   VAR_INPUT
      "string" : String;
      part_names : Array[0..19] of String;
   END_VAR
   VAR_OUTPUT
      true : Bool;
   END_VAR
BEGIN

REGION Network 1
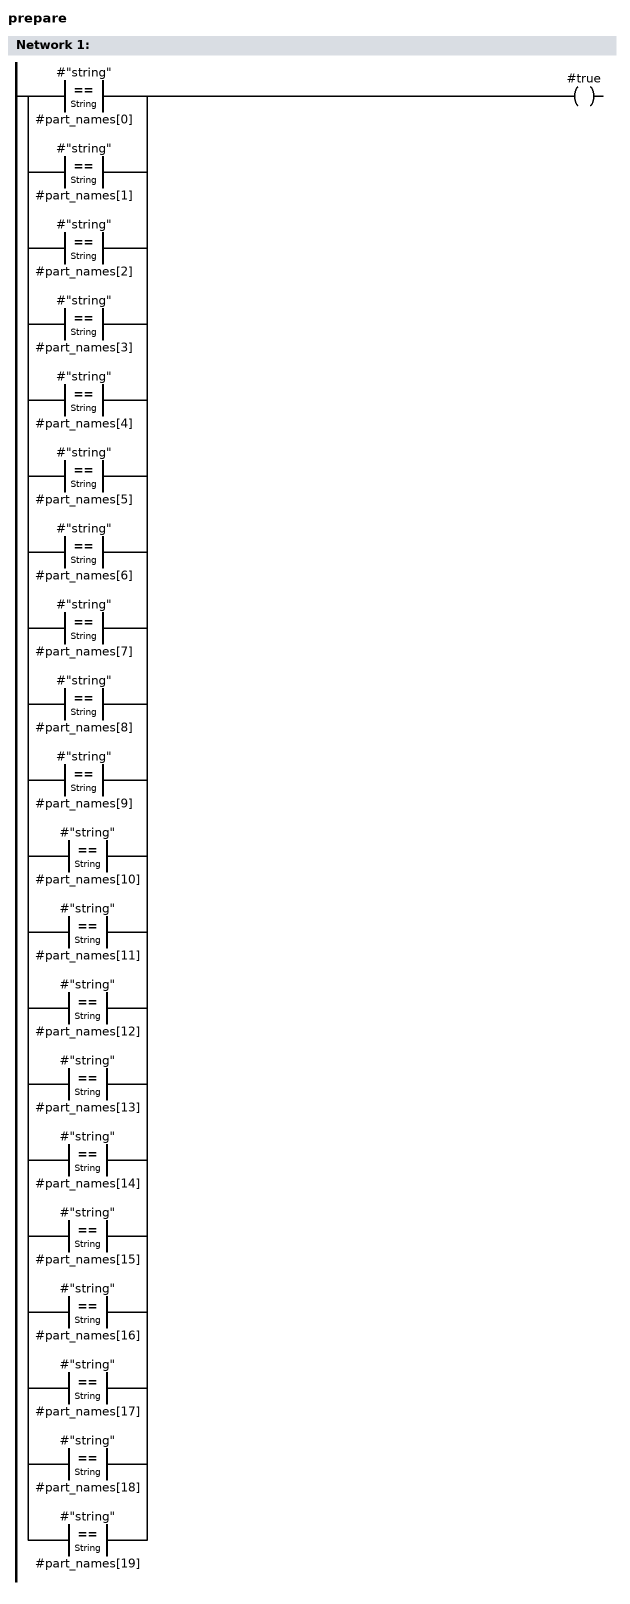
   RUNG wire#powerrail
      { S7_Templates := "SrcType := String" } EQ_Contact(in1 := #"string", in2 := #part_names[0])
      wire#w1
      Coil( #true )
   END_RUNG
   RUNG wire#powerrail
      { S7_Templates := "SrcType := String" } EQ_Contact(in1 := #"string", in2 := #part_names[1])
   END_RUNG wire#w1
   RUNG wire#powerrail
      { S7_Templates := "SrcType := String" } EQ_Contact(in1 := #"string", in2 := #part_names[2])
   END_RUNG wire#w1
   RUNG wire#powerrail
      { S7_Templates := "SrcType := String" } EQ_Contact(in1 := #"string", in2 := #part_names[3])
   END_RUNG wire#w1
   RUNG wire#powerrail
      { S7_Templates := "SrcType := String" } EQ_Contact(in1 := #"string", in2 := #part_names[4])
   END_RUNG wire#w1
   RUNG wire#powerrail
      { S7_Templates := "SrcType := String" } EQ_Contact(in1 := #"string", in2 := #part_names[5])
   END_RUNG wire#w1
   RUNG wire#powerrail
      { S7_Templates := "SrcType := String" } EQ_Contact(in1 := #"string", in2 := #part_names[6])
   END_RUNG wire#w1
   RUNG wire#powerrail
      { S7_Templates := "SrcType := String" } EQ_Contact(in1 := #"string", in2 := #part_names[7])
   END_RUNG wire#w1
   RUNG wire#powerrail
      { S7_Templates := "SrcType := String" } EQ_Contact(in1 := #"string", in2 := #part_names[8])
   END_RUNG wire#w1
   RUNG wire#powerrail
      { S7_Templates := "SrcType := String" } EQ_Contact(in1 := #"string", in2 := #part_names[9])
   END_RUNG wire#w1
   RUNG wire#powerrail
      { S7_Templates := "SrcType := String" } EQ_Contact(in1 := #"string", in2 := #part_names[10])
   END_RUNG wire#w1
   RUNG wire#powerrail
      { S7_Templates := "SrcType := String" } EQ_Contact(in1 := #"string", in2 := #part_names[11])
   END_RUNG wire#w1
   RUNG wire#powerrail
      { S7_Templates := "SrcType := String" } EQ_Contact(in1 := #"string", in2 := #part_names[12])
   END_RUNG wire#w1
   RUNG wire#powerrail
      { S7_Templates := "SrcType := String" } EQ_Contact(in1 := #"string", in2 := #part_names[13])
   END_RUNG wire#w1
   RUNG wire#powerrail
      { S7_Templates := "SrcType := String" } EQ_Contact(in1 := #"string", in2 := #part_names[14])
   END_RUNG wire#w1
   RUNG wire#powerrail
      { S7_Templates := "SrcType := String" } EQ_Contact(in1 := #"string", in2 := #part_names[15])
   END_RUNG wire#w1
   RUNG wire#powerrail
      { S7_Templates := "SrcType := String" } EQ_Contact(in1 := #"string", in2 := #part_names[16])
   END_RUNG wire#w1
   RUNG wire#powerrail
      { S7_Templates := "SrcType := String" } EQ_Contact(in1 := #"string", in2 := #part_names[17])
   END_RUNG wire#w1
   RUNG wire#powerrail
      { S7_Templates := "SrcType := String" } EQ_Contact(in1 := #"string", in2 := #part_names[18])
   END_RUNG wire#w1
   RUNG wire#powerrail
      { S7_Templates := "SrcType := String" } EQ_Contact(in1 := #"string", in2 := #part_names[19])
   END_RUNG wire#w1
   // the same network as SCL:
   #true := (#"string" = #part_names[0]) OR (#"string" = #part_names[1]) OR (#"string" = #part_names[2]) OR (#"string" = #part_names[3]) OR (#"string" = #part_names[4]) OR (#"string" = #part_names[5]) OR (#"string" = #part_names[6]) OR (#"string" = #part_names[7]) OR (#"string" = #part_names[8]) OR (#"string" = #part_names[9]) OR (#"string" = #part_names[10]) OR (#"string" = #part_names[11]) OR (#"string" = #part_names[12]) OR (#"string" = #part_names[13]) OR (#"string" = #part_names[14]) OR (#"string" = #part_names[15]) OR (#"string" = #part_names[16]) OR (#"string" = #part_names[17]) OR (#"string" = #part_names[18]) OR (#"string" = #part_names[19]);
END_REGION
END_FUNCTION_BLOCK

ORGANIZATION_BLOCK "Main"   // OB1, LAD, ProgramCycle
TITLE = "Main Program Sweep (Cycle)"
{ S7_Optimized_Access := 'TRUE' }
VERSION : 0.1
   VAR_INPUT
      Initial_Call : Bool;   // Initial call of this OB
      Remanence : Bool;   // =True, if remanent data are available
   END_VAR
   VAR_TEMP   // added for the SCL form of the ladder/FBD networks
      _w1 : Bool;
   END_VAR
BEGIN

REGION Network 1
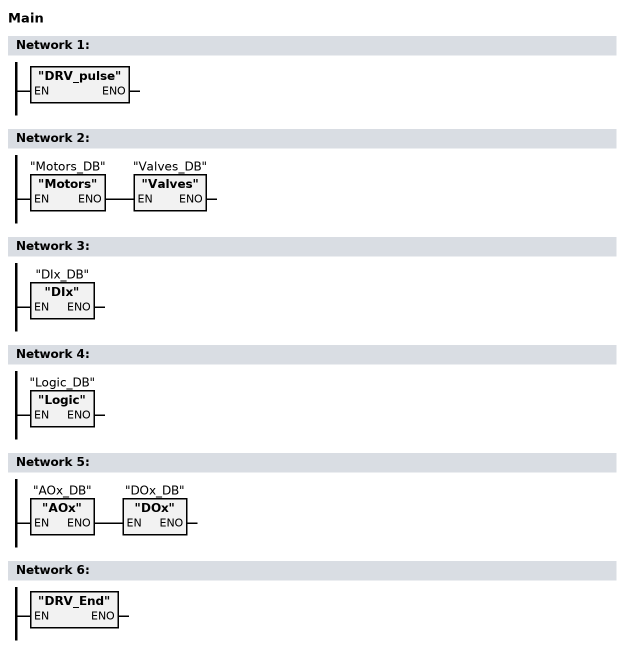
   RUNG wire#powerrail
      "DRV_pulse"()
   END_RUNG
   // the same network as SCL:
   "DRV_pulse"();
END_REGION

REGION Network 2
   RUNG wire#powerrail
      "Motors_DB"()
      "Valves_DB"()
   END_RUNG
   // the same network as SCL:
   "Motors_DB"(ENO => #_w1);   // "Motors"
   IF #_w1 THEN
       "Valves_DB"();   // "Valves"
   END_IF;
END_REGION

REGION Network 3
   RUNG wire#powerrail
      "DIx_DB"()
   END_RUNG
   // the same network as SCL:
   "DIx_DB"();   // "DIx"
END_REGION

REGION Network 4
   RUNG wire#powerrail
      "Logic_DB"()
   END_RUNG
   // the same network as SCL:
   "Logic_DB"();   // "Logic"
END_REGION

REGION Network 5
   RUNG wire#powerrail
      "AOx_DB"()
      "DOx_DB"()
   END_RUNG
   // the same network as SCL:
   "AOx_DB"(ENO => #_w1);   // "AOx"
   IF #_w1 THEN
       "DOx_DB"();   // "DOx"
   END_IF;
END_REGION

REGION Network 6
   RUNG wire#powerrail
      "DRV_End"()
   END_RUNG
   // the same network as SCL:
   "DRV_End"();
END_REGION
END_ORGANIZATION_BLOCK

// folder: DRV_Devices

FUNCTION_BLOCK "DRV_M_D"   // FB110, LAD
{ S7_Optimized_Access := 'FALSE' }
VERSION : 0.1
   VAR_INPUT
      FB_QF : Bool;   // защитный автомат / Защитный автомат
      FB_KM : Bool;   // привод запущен / Пускатель
      FB_Service : Bool;   // авария частотника / Сервисный выключатель
      FB_Termo : Bool;   // Термозащита
      FB_Alarm : Bool;   // Внешняя авария
      All_Block : Bool;   // Аварийный останов
   END_VAR
   VAR_OUTPUT
      Signal : Bool;   // Команда запуска двигателя
   END_VAR
   VAR_IN_OUT
      S_Alarm : Bool;   // Наличие аварии
   END_VAR
   VAR
      CMD : Struct   // Основные команды / Блок команд
         Hand : Bool;   // 0 - авто, 1 - ручной / 0 - Авто, 1 - Ручной
         Start_A : Bool;   // Автозапуск / Запуск в авторежиме
         Start_M : Bool;   // Ручной - вперёд / Запуск в ручном режиме
         Force : Bool;   // Принудительный
         Lock : Bool;   // Блокировать / Блокировка
         Local : Bool;   // Локальный
         Service : Bool;   // Сервис
         Safety : Bool;   // Безопасность
         Alarm : Bool;   // Есть авария / Авария
         Reset : Bool;   // Сброс аварий
         Sim : Bool;   // Режим симуляции
      END_STRUCT;
      Mode : Int;   // Режим работы
      Status : Int;   // Статус устройства
      Use : Struct   // Функционал
         Ready : Bool := true;   // Готовность
         QF : Bool := true;   // Защитный автомат
         KM : Bool := true;   // Пускатель
         Serivce : Bool;   // Сервисный выключатель
         Termo : Bool;   // Термозащита
         Alarm : Bool;   // Внешняя авария
      END_STRUCT;
      FB : Struct   // Функционал
         Ready : Bool;   // Готовность к запуску
         QF : Bool;   // Защитный автомат
         KM : Bool;   // Пускатель
         Serivce : Bool;   // Сервисный выключатель
         Termo : Bool;   // Термозащита
         Alarm : Bool;   // Внешняя авария
      END_STRUCT;
      Go : Bool;   // Запуск
      ON : Bool;   // Успешно запущено
      OFF : Bool;   // Успешно остановлено
      G_Sim_On : Bool;   // Запуск глобальной симуляции
      G_Sim_Off : Bool;   // Отключение глобальной симуляции
      Wait_On : Struct   // Ожидание ОС контактора / Время на запуск
         SP : Int := 2;
         Now : Int;
         "Exit" : Bool;
         Start : Bool;
         Pause : Bool;
         Reset : Bool;   // Сброс таймера
      END_STRUCT;
      Wait_Off : Struct   // Ожидание концевиков / Время на останов
         SP : Int := 2;
         Now : Int;
         "Exit" : Bool;
         Start : Bool;
         Pause : Bool;
         Reset : Bool;   // Сброс таймера
      END_STRUCT;
      Inv : Struct   // Инверсия сигналов
         Reserv : Bool;
         QF : Bool;   // Защитный автомат
         KM : Bool;   // Пускатель
         Serivce : Bool;   // Сервисный выключатель
         Termo : Bool;   // Термозащита
         Alarm : Bool;   // Внешняя авария
      END_STRUCT;
      Alm : Struct   // Сбор аварий / Список аварий
         Block : Bool;   // Аварийная остановка
         QF : Bool;   // привод не готов / Выбило защитный автомат
         Start : Bool;   // Ошибка при запуске
         Stop : Bool;   // Ошибка при останове
         PTC : Bool;   // термозащита / Сработала термозащита
         Alarm : Bool;   // Внешняя авария
         Safety : Bool;   // Сработала безопасность
      END_STRUCT;
      Alarm : Word;   // Слово аварий
      Res_h : DInt;   // наработка (ч)
      Res_s : DInt;   // наработка (с)
   END_VAR
   VAR_TEMP   // added for the SCL form of the ladder/FBD networks
      _w1 : Bool;
      _w2 : Bool;
   END_VAR
BEGIN

REGION Network 1: Режим глобальной симуляции
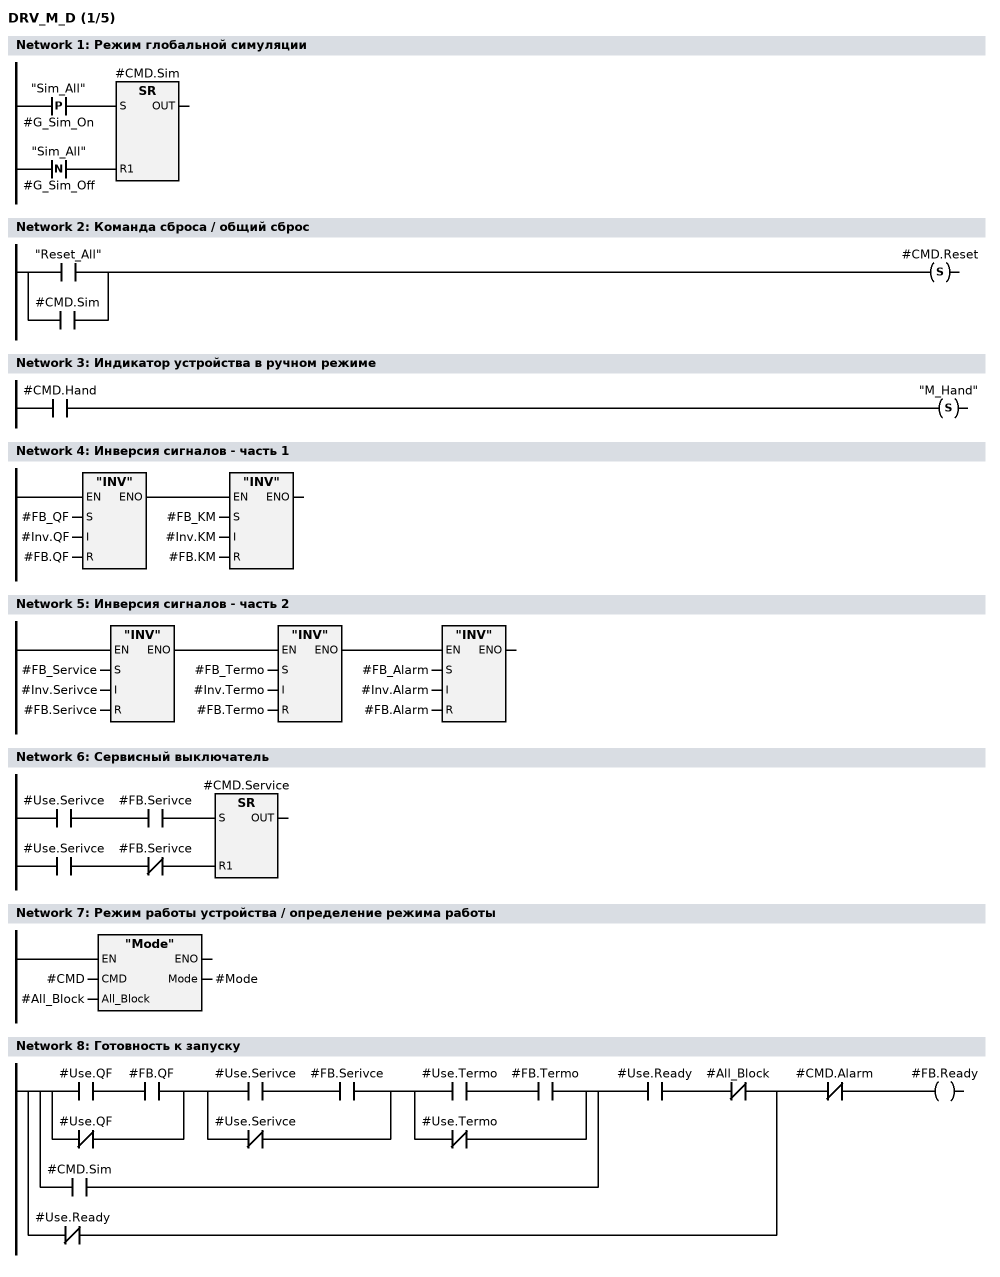
   RUNG wire#powerrail
      P_Contact(operand := "Sim_All", bit := #G_Sim_On)
      S_SR(operand := #CMD.Sim, r1 := wire#w1)
   END_RUNG
   RUNG wire#powerrail
      N_Contact(operand := "Sim_All", bit := #G_Sim_Off)
   END_RUNG wire#w1
   // the same network as SCL:
   #_w1 := "Sim_All" AND NOT #G_Sim_On;   // rising edge of "Sim_All"
   #G_Sim_On := "Sim_All";
   #_w2 := NOT "Sim_All" AND #G_Sim_Off;   // falling edge of "Sim_All"
   #G_Sim_Off := "Sim_All";
   IF #_w1 THEN
       #CMD.Sim := TRUE;   // SR flip-flop
   END_IF;
   IF #_w2 THEN #CMD.Sim := FALSE; END_IF;
END_REGION

REGION Network 2: Команда сброса / общий сброс
   RUNG wire#powerrail
      Contact( "Reset_All" )
      wire#w1
      S_Coil( #CMD.Reset )
   END_RUNG
   RUNG wire#powerrail
      Contact( #CMD.Sim )
   END_RUNG wire#w1
   // the same network as SCL:
   IF "Reset_All" OR #CMD.Sim THEN #CMD.Reset := TRUE; END_IF;
END_REGION

REGION Network 3: Индикатор устройства в ручном режиме
   RUNG wire#powerrail
      Contact( #CMD.Hand )
      S_Coil( "M_Hand" )
   END_RUNG
   // the same network as SCL:
   IF #CMD.Hand THEN "M_Hand" := TRUE; END_IF;
END_REGION

REGION Network 4: Инверсия сигналов - часть 1
   RUNG wire#powerrail
      "INV"(S := #FB_QF, I := #Inv.QF, R := #FB.QF)
      "INV"(S := #FB_KM, I := #Inv.KM, R := #FB.KM)
   END_RUNG
   // the same network as SCL:
   "INV"(S := #FB_QF, I := #Inv.QF, R := #FB.QF, ENO => #_w1);
   IF #_w1 THEN "INV"(S := #FB_KM, I := #Inv.KM, R := #FB.KM); END_IF;
END_REGION

REGION Network 5: Инверсия сигналов - часть 2
   RUNG wire#powerrail
      "INV"(S := #FB_Service, I := #Inv.Serivce, R := #FB.Serivce)
      "INV"(S := #FB_Termo, I := #Inv.Termo, R := #FB.Termo)
      "INV"(S := #FB_Alarm, I := #Inv.Alarm, R := #FB.Alarm)
   END_RUNG
   // the same network as SCL:
   "INV"(S := #FB_Service, I := #Inv.Serivce, R := #FB.Serivce, ENO => #_w1);
   "INV"(EN := #_w1, S := #FB_Termo, I := #Inv.Termo, R := #FB.Termo, ENO => #_w2);
   IF #_w2 THEN "INV"(S := #FB_Alarm, I := #Inv.Alarm, R := #FB.Alarm); END_IF;
END_REGION

REGION Network 6: Сервисный выключатель
   RUNG wire#powerrail
      Contact( #Use.Serivce )
      Contact( #FB.Serivce )
      S_SR(operand := #CMD.Service, r1 := wire#w1)
   END_RUNG
   RUNG wire#powerrail
      Contact( #Use.Serivce )
      I_Contact( #FB.Serivce )
   END_RUNG wire#w1
   // the same network as SCL:
   IF #Use.Serivce AND #FB.Serivce THEN
       #CMD.Service := TRUE;   // SR flip-flop
   END_IF;
   IF #Use.Serivce AND NOT #FB.Serivce THEN #CMD.Service := FALSE; END_IF;
END_REGION

REGION Network 7: Режим работы устройства / определение режима работы
   RUNG wire#powerrail
      "Mode"(CMD := #CMD, All_Block := #All_Block, Mode => #Mode)
   END_RUNG
   // the same network as SCL:
   "Mode"(CMD := #CMD, All_Block := #All_Block, Mode => #Mode);
END_REGION

REGION Network 8: Готовность к запуску
   RUNG wire#powerrail
      Contact( #Use.QF )
      Contact( #FB.QF )
      wire#w1
      Contact( #Use.Serivce )
      Contact( #FB.Serivce )
      wire#w2
      Contact( #Use.Termo )
      Contact( #FB.Termo )
      wire#w3
      Contact( #Use.Ready )
      I_Contact( #All_Block )
      wire#w4
      I_Contact( #CMD.Alarm )
      Coil( #FB.Ready )
   END_RUNG
   RUNG wire#powerrail
      I_Contact( #Use.QF )
   END_RUNG wire#w1
   RUNG wire#w1
      I_Contact( #Use.Serivce )
   END_RUNG wire#w2
   RUNG wire#w2
      I_Contact( #Use.Termo )
   END_RUNG wire#w3
   RUNG wire#powerrail
      Contact( #CMD.Sim )
   END_RUNG wire#w3
   RUNG wire#powerrail
      I_Contact( #Use.Ready )
   END_RUNG wire#w4
   // the same network as SCL:
   #FB.Ready := ((((((#Use.QF AND #FB.QF) OR NOT #Use.QF) AND ((#Use.Serivce AND #FB.Serivce) OR NOT #Use.Serivce) AND ((#Use.Termo AND #FB.Termo) OR NOT #Use.Termo)) OR #CMD.Sim) AND #Use.Ready AND NOT #All_Block) OR NOT #Use.Ready) AND NOT #CMD.Alarm;
END_REGION

REGION Network 9: Управление запуском / дискретный управляющий сигнал
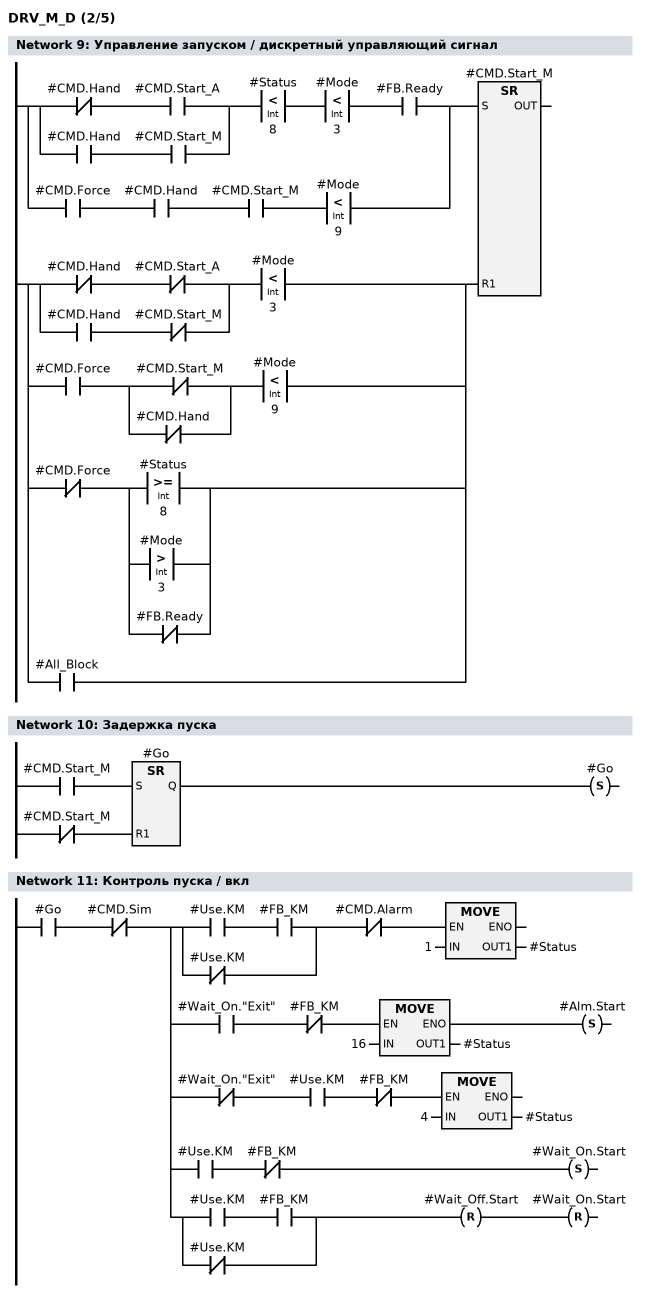
   RUNG wire#powerrail
      I_Contact( #CMD.Hand )
      Contact( #CMD.Start_A )
      wire#w1
      { S7_Templates := "SrcType := Int" } LT_Contact(in1 := #Status, in2 := 8)
      { S7_Templates := "SrcType := Int" } LT_Contact(in1 := #Mode, in2 := 3)
      Contact( #FB.Ready )
      wire#w2
      S_SR(operand := #CMD.Start_M, r1 := wire#w7)
   END_RUNG
   RUNG wire#powerrail
      Contact( #CMD.Hand )
      Contact( #CMD.Start_M )
   END_RUNG wire#w1
   RUNG wire#powerrail
      Contact( #CMD.Force )
      Contact( #CMD.Hand )
      Contact( #CMD.Start_M )
      { S7_Templates := "SrcType := Int" } LT_Contact(in1 := #Mode, in2 := 9)
   END_RUNG wire#w2
   RUNG wire#powerrail
      I_Contact( #CMD.Hand )
      I_Contact( #CMD.Start_A )
      wire#w3
      { S7_Templates := "SrcType := Int" } LT_Contact(in1 := #Mode, in2 := 3)
   END_RUNG wire#w7
   RUNG wire#powerrail
      Contact( #CMD.Hand )
      I_Contact( #CMD.Start_M )
   END_RUNG wire#w3
   RUNG wire#powerrail
      Contact( #CMD.Force )
      wire#w4
      I_Contact( #CMD.Start_M )
      wire#w5
      { S7_Templates := "SrcType := Int" } LT_Contact(in1 := #Mode, in2 := 9)
   END_RUNG wire#w7
   RUNG wire#w4
      I_Contact( #CMD.Hand )
   END_RUNG wire#w5
   RUNG wire#powerrail
      I_Contact( #CMD.Force )
      wire#w6
      { S7_Templates := "SrcType := Int" } GE_Contact(in1 := #Status, in2 := 8)
   END_RUNG wire#w7
   RUNG wire#w6
      { S7_Templates := "SrcType := Int" } GT_Contact(in1 := #Mode, in2 := 3)
   END_RUNG wire#w7
   RUNG wire#w6
      I_Contact( #FB.Ready )
   END_RUNG wire#w7
   RUNG wire#powerrail
      Contact( #All_Block )
   END_RUNG wire#w7
   // the same network as SCL:
   #_w1 := (((NOT #CMD.Hand AND NOT #CMD.Start_A) OR (#CMD.Hand AND NOT #CMD.Start_M)) AND (#Mode < 3)) OR (#CMD.Force AND (NOT #CMD.Start_M OR NOT #CMD.Hand) AND (#Mode < 9)) OR (NOT #CMD.Force AND ((#Status >= 8) OR (#Mode > 3) OR NOT #FB.Ready)) OR #All_Block;
   IF (((NOT #CMD.Hand AND #CMD.Start_A) OR (#CMD.Hand AND #CMD.Start_M)) AND (#Status < 8) AND (#Mode < 3) AND #FB.Ready) OR (#CMD.Force AND #CMD.Hand AND #CMD.Start_M AND (#Mode < 9)) THEN
       #CMD.Start_M := TRUE;   // SR flip-flop
   END_IF;
   IF #_w1 THEN #CMD.Start_M := FALSE; END_IF;
END_REGION

REGION Network 10: Задержка пуска
   RUNG wire#powerrail
      Contact( #CMD.Start_M )
      S_SR(operand := #Go, r1 := wire#w1)
      S_Coil( #Go )
   END_RUNG
   RUNG wire#powerrail
      I_Contact( #CMD.Start_M )
   END_RUNG wire#w1
   // the same network as SCL:
   IF #CMD.Start_M THEN
       #Go := TRUE;   // SR flip-flop
   END_IF;
   IF NOT #CMD.Start_M THEN #Go := FALSE; END_IF;
   IF #Go THEN #Go := TRUE; END_IF;
END_REGION

REGION Network 11: Контроль пуска / вкл
   RUNG wire#powerrail
      Contact( #Go )
      I_Contact( #CMD.Sim )
      wire#w1
      Contact( #Use.KM )
      Contact( #FB_KM )
      wire#w2
      I_Contact( #CMD.Alarm )
      { S7_GenerateENO := "TRUE" } Move(in := 1, out1 => #Status)
   END_RUNG
   RUNG wire#w1
      I_Contact( #Use.KM )
   END_RUNG wire#w2
   RUNG wire#w1
      Contact( #Wait_On."Exit" )
      I_Contact( #FB_KM )
      { S7_GenerateENO := "TRUE" } Move(in := 16, out1 => #Status)
      S_Coil( #Alm.Start )
   END_RUNG
   RUNG wire#w1
      I_Contact( #Wait_On."Exit" )
      Contact( #Use.KM )
      I_Contact( #FB_KM )
      { S7_GenerateENO := "TRUE" } Move(in := 4, out1 => #Status)
   END_RUNG
   RUNG wire#w1
      Contact( #Use.KM )
      I_Contact( #FB_KM )
      S_Coil( #Wait_On.Start )
   END_RUNG
   RUNG wire#w1
      Contact( #Use.KM )
      Contact( #FB_KM )
      wire#w3
      R_Coil( #Wait_Off.Start )
      R_Coil( #Wait_On.Start )
   END_RUNG
   RUNG wire#w1
      I_Contact( #Use.KM )
   END_RUNG wire#w3
   // the same network as SCL:
   // ENO of a box is taken as its EN; it also drops when the box reports an error
   #_w1 := #Go AND NOT #CMD.Sim;
   IF #_w1 AND ((#Use.KM AND #FB_KM) OR NOT #Use.KM) AND NOT #CMD.Alarm THEN #Status := 1; END_IF;
   IF #_w1 AND #Wait_On."Exit" AND NOT #FB_KM THEN
       #Status := 16;
       #Alm.Start := TRUE;
   END_IF;
   IF #_w1 AND NOT #Wait_On."Exit" AND #Use.KM AND NOT #FB_KM THEN #Status := 4; END_IF;
   IF #_w1 AND #Use.KM AND NOT #FB_KM THEN #Wait_On.Start := TRUE; END_IF;
   IF #_w1 AND ((#Use.KM AND #FB_KM) OR NOT #Use.KM) THEN
       #Wait_Off.Start := FALSE;
       #Wait_On.Start := FALSE;
   END_IF;
END_REGION

REGION Network 12: Контроль останова / выкл
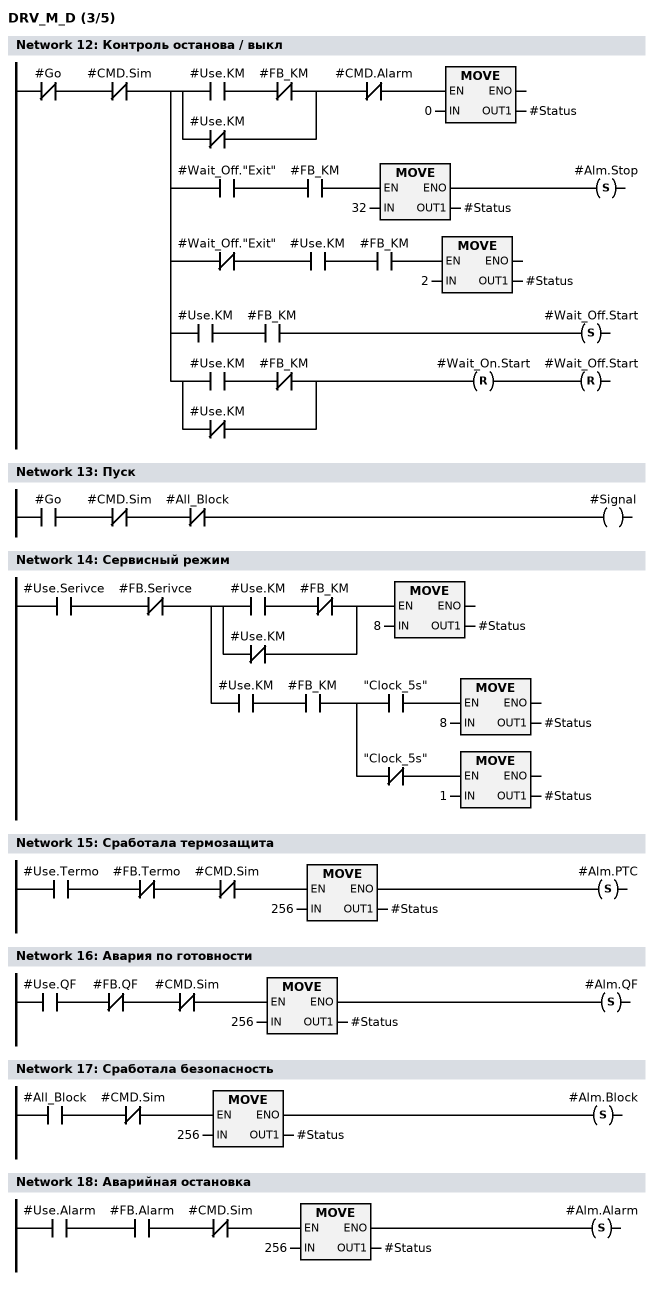
   RUNG wire#powerrail
      I_Contact( #Go )
      I_Contact( #CMD.Sim )
      wire#w1
      Contact( #Use.KM )
      I_Contact( #FB_KM )
      wire#w2
      I_Contact( #CMD.Alarm )
      { S7_GenerateENO := "TRUE" } Move(in := 0, out1 => #Status)
   END_RUNG
   RUNG wire#w1
      I_Contact( #Use.KM )
   END_RUNG wire#w2
   RUNG wire#w1
      Contact( #Wait_Off."Exit" )
      Contact( #FB_KM )
      { S7_GenerateENO := "TRUE" } Move(in := 32, out1 => #Status)
      S_Coil( #Alm.Stop )
   END_RUNG
   RUNG wire#w1
      I_Contact( #Wait_Off."Exit" )
      Contact( #Use.KM )
      Contact( #FB_KM )
      { S7_GenerateENO := "TRUE" } Move(in := 2, out1 => #Status)
   END_RUNG
   RUNG wire#w1
      Contact( #Use.KM )
      Contact( #FB_KM )
      S_Coil( #Wait_Off.Start )
   END_RUNG
   RUNG wire#w1
      Contact( #Use.KM )
      I_Contact( #FB_KM )
      wire#w3
      R_Coil( #Wait_On.Start )
      R_Coil( #Wait_Off.Start )
   END_RUNG
   RUNG wire#w1
      I_Contact( #Use.KM )
   END_RUNG wire#w3
   // the same network as SCL:
   // ENO of a box is taken as its EN; it also drops when the box reports an error
   #_w1 := NOT #Go AND NOT #CMD.Sim;
   IF #_w1 AND ((#Use.KM AND NOT #FB_KM) OR NOT #Use.KM) AND NOT #CMD.Alarm THEN #Status := 0; END_IF;
   IF #_w1 AND #Wait_Off."Exit" AND #FB_KM THEN
       #Status := 32;
       #Alm.Stop := TRUE;
   END_IF;
   IF #_w1 AND NOT #Wait_Off."Exit" AND #Use.KM AND #FB_KM THEN #Status := 2; END_IF;
   IF #_w1 AND #Use.KM AND #FB_KM THEN #Wait_Off.Start := TRUE; END_IF;
   IF #_w1 AND ((#Use.KM AND NOT #FB_KM) OR NOT #Use.KM) THEN
       #Wait_On.Start := FALSE;
       #Wait_Off.Start := FALSE;
   END_IF;
END_REGION

REGION Network 13: Пуск
   RUNG wire#powerrail
      Contact( #Go )
      I_Contact( #CMD.Sim )
      I_Contact( #All_Block )
      Coil( #Signal )
   END_RUNG
   // the same network as SCL:
   #Signal := #Go AND NOT #CMD.Sim AND NOT #All_Block;
END_REGION

REGION Network 14: Сервисный режим
   RUNG wire#powerrail
      Contact( #Use.Serivce )
      I_Contact( #FB.Serivce )
      wire#w1
      Contact( #Use.KM )
      I_Contact( #FB_KM )
      wire#w2
      Move(in := 8, out1 => #Status)
   END_RUNG
   RUNG wire#w1
      I_Contact( #Use.KM )
   END_RUNG wire#w2
   RUNG wire#w1
      Contact( #Use.KM )
      Contact( #FB_KM )
      wire#w3
      Contact( "Clock_5s" )
      Move(in := 8, out1 => #Status)
   END_RUNG
   RUNG wire#w3
      I_Contact( "Clock_5s" )
      Move(in := 1, out1 => #Status)
   END_RUNG
   // the same network as SCL:
   #_w1 := #Use.Serivce AND NOT #FB.Serivce;
   IF #_w1 AND ((#Use.KM AND NOT #FB_KM) OR NOT #Use.KM) THEN #Status := 8; END_IF;
   #_w2 := #_w1 AND #Use.KM AND #FB_KM;
   IF #_w2 AND "Clock_5s" THEN #Status := 8; END_IF;
   IF #_w2 AND NOT "Clock_5s" THEN #Status := 1; END_IF;
END_REGION

REGION Network 15: Сработала термозащита
   RUNG wire#powerrail
      Contact( #Use.Termo )
      I_Contact( #FB.Termo )
      I_Contact( #CMD.Sim )
      { S7_GenerateENO := "TRUE" } Move(in := 256, out1 => #Status)
      S_Coil( #Alm.PTC )
   END_RUNG
   // the same network as SCL:
   // ENO of a box is taken as its EN; it also drops when the box reports an error
   IF #Use.Termo AND NOT #FB.Termo AND NOT #CMD.Sim THEN
       #Status := 256;
       #Alm.PTC := TRUE;
   END_IF;
END_REGION

REGION Network 16: Авария по готовности
   RUNG wire#powerrail
      Contact( #Use.QF )
      I_Contact( #FB.QF )
      I_Contact( #CMD.Sim )
      { S7_GenerateENO := "TRUE" } Move(in := 256, out1 => #Status)
      S_Coil( #Alm.QF )
   END_RUNG
   // the same network as SCL:
   // ENO of a box is taken as its EN; it also drops when the box reports an error
   IF #Use.QF AND NOT #FB.QF AND NOT #CMD.Sim THEN
       #Status := 256;
       #Alm.QF := TRUE;
   END_IF;
END_REGION

REGION Network 17: Сработала безопасность
   RUNG wire#powerrail
      Contact( #All_Block )
      I_Contact( #CMD.Sim )
      { S7_GenerateENO := "TRUE" } Move(in := 256, out1 => #Status)
      S_Coil( #Alm.Block )
   END_RUNG
   // the same network as SCL:
   // ENO of a box is taken as its EN; it also drops when the box reports an error
   IF #All_Block AND NOT #CMD.Sim THEN
       #Status := 256;
       #Alm.Block := TRUE;
   END_IF;
END_REGION

REGION Network 18: Аварийная остановка
   RUNG wire#powerrail
      Contact( #Use.Alarm )
      Contact( #FB.Alarm )
      I_Contact( #CMD.Sim )
      { S7_GenerateENO := "TRUE" } Move(in := 256, out1 => #Status)
      S_Coil( #Alm.Alarm )
   END_RUNG
   // the same network as SCL:
   // ENO of a box is taken as its EN; it also drops when the box reports an error
   IF #Use.Alarm AND #FB.Alarm AND NOT #CMD.Sim THEN
       #Status := 256;
       #Alm.Alarm := TRUE;
   END_IF;
END_REGION

REGION Network 19: Сигнал аварии
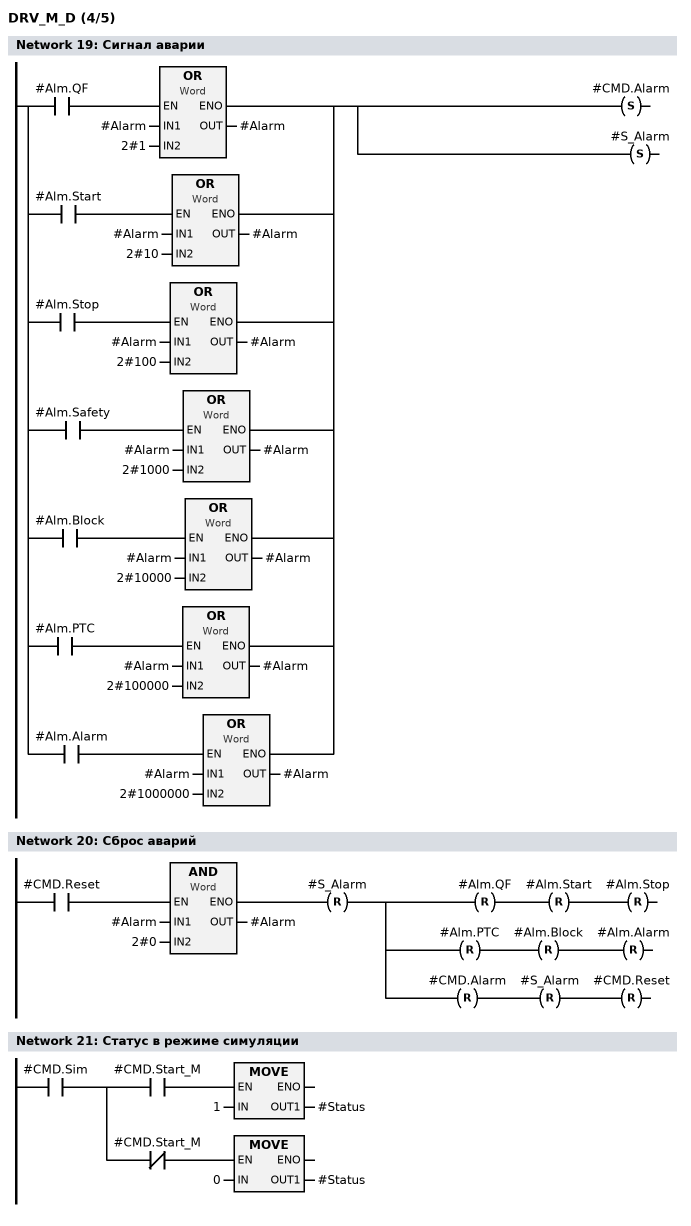
   // no checked SCL form for this network; see the picture
END_REGION

REGION Network 20: Сброс аварий
   // no checked SCL form for this network; see the picture
END_REGION

REGION Network 21: Статус в режиме симуляции
   RUNG wire#powerrail
      Contact( #CMD.Sim )
      wire#w1
      Contact( #CMD.Start_M )
      { S7_GenerateENO := "TRUE" } Move(in := 1, out1 => #Status)
   END_RUNG
   RUNG wire#w1
      I_Contact( #CMD.Start_M )
      { S7_GenerateENO := "TRUE" } Move(in := 0, out1 => #Status)
   END_RUNG
   // the same network as SCL:
   IF #CMD.Sim AND #CMD.Start_M THEN #Status := 1; END_IF;
   IF #CMD.Sim AND NOT #CMD.Start_M THEN #Status := 0; END_IF;
END_REGION

REGION Network 22: Статус в локальным режиме
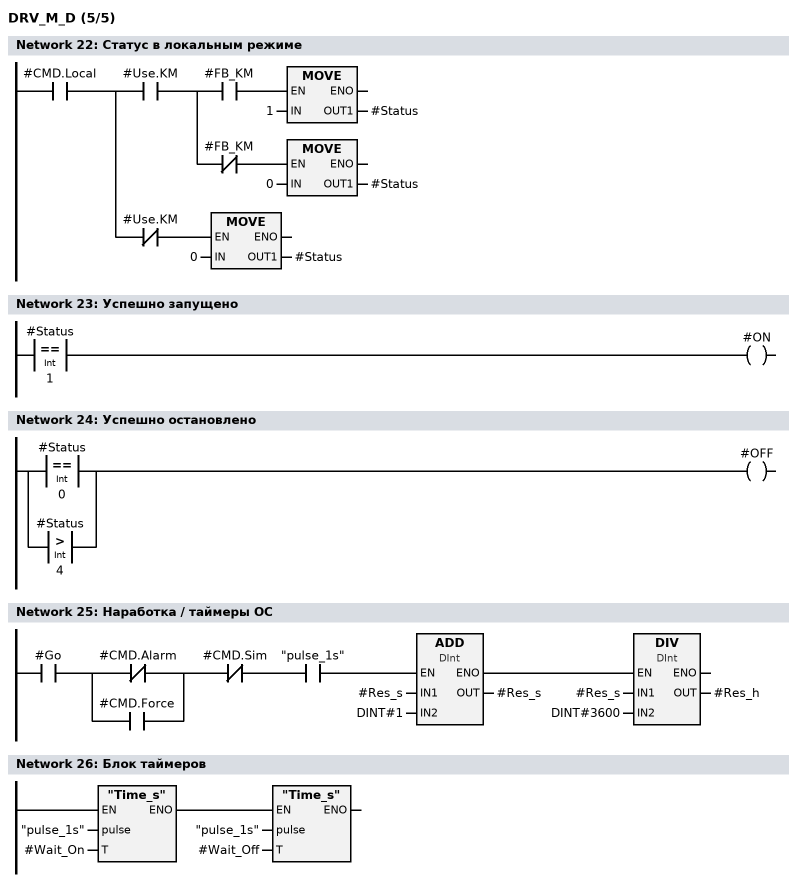
   RUNG wire#powerrail
      Contact( #CMD.Local )
      wire#w1
      Contact( #Use.KM )
      wire#w2
      Contact( #FB_KM )
      { S7_GenerateENO := "TRUE" } Move(in := 1, out1 => #Status)
   END_RUNG
   RUNG wire#w2
      I_Contact( #FB_KM )
      { S7_GenerateENO := "TRUE" } Move(in := 0, out1 => #Status)
   END_RUNG
   RUNG wire#w1
      I_Contact( #Use.KM )
      { S7_GenerateENO := "TRUE" } Move(in := 0, out1 => #Status)
   END_RUNG
   // the same network as SCL:
   #_w1 := #CMD.Local AND #Use.KM;
   IF #_w1 AND #FB_KM THEN #Status := 1; END_IF;
   IF #_w1 AND NOT #FB_KM THEN #Status := 0; END_IF;
   IF #CMD.Local AND NOT #Use.KM THEN #Status := 0; END_IF;
END_REGION

REGION Network 23: Успешно запущено
   RUNG wire#powerrail
      { S7_Templates := "SrcType := Int" } EQ_Contact(in1 := #Status, in2 := 1)
      Coil( #ON )
   END_RUNG
   // the same network as SCL:
   #ON := #Status = 1;
END_REGION

REGION Network 24: Успешно остановлено
   RUNG wire#powerrail
      { S7_Templates := "SrcType := Int" } EQ_Contact(in1 := #Status, in2 := 0)
      wire#w1
      Coil( #OFF )
   END_RUNG
   RUNG wire#powerrail
      { S7_Templates := "SrcType := Int" } GT_Contact(in1 := #Status, in2 := 4)
   END_RUNG wire#w1
   // the same network as SCL:
   #OFF := (#Status = 0) OR (#Status > 4);
END_REGION

REGION Network 25: Наработка / таймеры ОС
   RUNG wire#powerrail
      Contact( #Go )
      wire#w1
      I_Contact( #CMD.Alarm )
      wire#w2
      I_Contact( #CMD.Sim )
      Contact( "pulse_1s" )
      { S7_Templates := "SrcType := DInt"; S7_GenerateENO := "TRUE" } Add(in1 := #Res_s, in2 := DINT#1, out => #Res_s)
      { S7_Templates := "SrcType := DInt"; S7_GenerateENO := "TRUE" } Div(in1 := #Res_s, in2 := DINT#3600, out => #Res_h)
   END_RUNG
   RUNG wire#w1
      Contact( #CMD.Force )
   END_RUNG wire#w2
   // the same network as SCL:
   // ENO of a box is taken as its EN; it also drops when the box reports an error
   IF #Go AND (NOT #CMD.Alarm OR #CMD.Force) AND NOT #CMD.Sim AND "pulse_1s" THEN
       #Res_s := #Res_s + DINT#1;
       #Res_h := #Res_s / DINT#3600;
   END_IF;
END_REGION

REGION Network 26: Блок таймеров
   RUNG wire#powerrail
      "Time_s"(pulse := "pulse_1s", T := #Wait_On)
      "Time_s"(pulse := "pulse_1s", T := #Wait_Off)
   END_RUNG
   // the same network as SCL:
   "Time_s"(pulse := "pulse_1s", T := #Wait_On, ENO => #_w1);
   IF #_w1 THEN "Time_s"(pulse := "pulse_1s", T := #Wait_Off); END_IF;
END_REGION
END_FUNCTION_BLOCK

FUNCTION_BLOCK "DRV_M_DA"   // FB111, LAD
{ S7_Optimized_Access := 'FALSE' }
VERSION : 0.1
   VAR_INPUT
      FB_QF : Bool;   // защитный автомат / Защитный автомат
      FB_KM : Bool;   // привод запущен / Пускатель
      FB_Alarm : Bool;   // Внешняя авария
      FB_Cut_KM : Bool;   // Отсечной пускатель
      FB_Safety : Bool;   // Безопасность
      FB_Service : Bool;   // авария частотника / Сервисный выключатель
      FB_Termo : Bool;   // Термозащита
      Local_Start : Bool;   // Локальный пуск
      Local_Stop : Bool;   // Локальный стоп
      All_Block : Bool;   // Аварийный останов
   END_VAR
   VAR_OUTPUT
      Signal : Bool;   // Команда запуска двигателя
      Cut_KM : Bool;   // Команда на отсечной пускатель
      Analog : Bool;   // Управление аналоговым выходом
      SP : Real;   // Уставка скорости
   END_VAR
   VAR_IN_OUT
      S_Alarm : Bool;   // Наличие аварии
   END_VAR
   VAR
      CMD : Struct   // Основные команды / Блок команд
         Hand : Bool;   // 0 - авто, 1 - ручной / 0 - Авто, 1 - Ручной
         Start_A : Bool;   // Автозапуск / Запуск в авторежиме
         Start_M : Bool;   // Ручной - вперёд / Запуск в ручном режиме
         Force : Bool;   // Принудительный
         Lock : Bool;   // Блокировать / Блокировка
         Local : Bool;   // Локальный
         Service : Bool;   // Сервис
         Safety : Bool;   // Безопасность
         Alarm : Bool;   // Есть авария / Авария
         Reset : Bool;   // Сброс аварий
         Sim : Bool;   // Режим симуляции
      END_STRUCT;
      Mode : Int;   // Режим работы
      Status : Int;   // Статус устройства
      Use : Struct   // Функционал
         Ready : Bool := true;   // Готовность
         QF : Bool := true;   // Защитный автомат
         KM : Bool := true;   // Пускатель
         Serivce : Bool;   // Сервисный выключатель
         Termo : Bool;   // Термозащита
         Alarm : Bool;   // Внешняя авария
         Safety : Bool;   // Безопасность
         Cut_KM : Bool;   // Отсечной пускатель
         Local_Keys : Bool;   // Локальное управление
         Analog : Bool := true;   // Управлять аналоговым выходом
      END_STRUCT;
      FB : Struct   // Функционал
         Ready : Bool;   // Готовность к запуску
         QF : Bool;   // Защитный автомат
         KM : Bool;   // Пускатель
         Serivce : Bool;   // Сервисный выключатель
         Termo : Bool;   // Термозащита
         Alarm : Bool;   // Внешняя авария
         Safety : Bool;   // Безопасность
         Cut_KM : Bool;   // Отсечной пускатель
         Local_Start : Bool;   // Локальный пуск
         Local_Stop : Bool;   // Локальный стоп
      END_STRUCT;
      Go : Bool;   // Запуск
      ON : Bool;   // Успешно запущено
      OFF : Bool;   // Успешно остановлено
      Cut_CMD : Bool;   // Запрос на включение отсечного пускателя
      G_Sim_On : Bool;   // Запуск глобальной симуляции
      G_Sim_Off : Bool;   // Отключение глобальной симуляции
      Wait_On : Struct   // Ожидание ОС контактора / Время на запуск
         SP : Int := 2;
         Now : Int;
         "Exit" : Bool;
         Start : Bool;
         Pause : Bool;
         Reset : Bool;   // Сброс таймера
      END_STRUCT;
      Wait_Off : Struct   // Ожидание концевиков / Время на останов
         SP : Int := 2;
         Now : Int;
         "Exit" : Bool;
         Start : Bool;
         Pause : Bool;
         Reset : Bool;   // Сброс таймера
      END_STRUCT;
      Delay_On : Struct   // Задержка пуска / Задержка запуска
         SP : Int := 0;
         Now : Int;
         "Exit" : Bool;
         Start : Bool;
         Pause : Bool;
         Reset : Bool;   // Сброс таймера
      END_STRUCT;
      Delay_Off : Struct   // Зажержка останова / Задержка останова
         SP : Int := 0;
         Now : Int;
         "Exit" : Bool;
         Start : Bool;
         Pause : Bool;
         Reset : Bool;   // Сброс таймера
      END_STRUCT;
      Inv : Struct   // Инверсия сигналов
         QF : Bool;   // Защитный автомат
         KM : Bool;   // Пускатель
         Serivce : Bool;   // Сервисный выключатель
         Termo : Bool;   // Термозащита
         Alarm : Bool;   // Внешняя авария
         Safety : Bool;   // Безопасность
         Cut_KM : Bool;   // Отсечной пускатель
         Local_Start : Bool;   // Локальный пуск
         Local_Stop : Bool;   // Локальный стоп
      END_STRUCT;
      Alm : Struct   // Сбор аварий / Список аварий
         Block : Bool;   // Аварийная остановка
         QF : Bool;   // привод не готов / Выбило защитный автомат
         Start : Bool;   // Ошибка при запуске
         Stop : Bool;   // Ошибка при останове
         PTC : Bool;   // термозащита / Сработала термозащита
         Alarm : Bool;   // Внешняя авария
         Safety : Bool;   // Сработала безопасность
         Cut_KM : Bool;   // Авария отсечного пускателя
      END_STRUCT;
      Alarm : Word;   // Слово аварий
      Res_h : DInt;   // наработка (ч)
      Res_s : DInt;   // наработка (с)
      SP_A : Real;   // Уставка скорости в авторежиме
      SP_M : Real;   // Уставка скорости в ручном режиме
      REQ_Cut_KM : "DRV_Micro";
   END_VAR
   VAR_TEMP   // added for the SCL form of the ladder/FBD networks
      _w1 : Bool;
      _w2 : Bool;
      _w3 : Bool;
   END_VAR
BEGIN

REGION Network 1: Режим глобальной симуляции
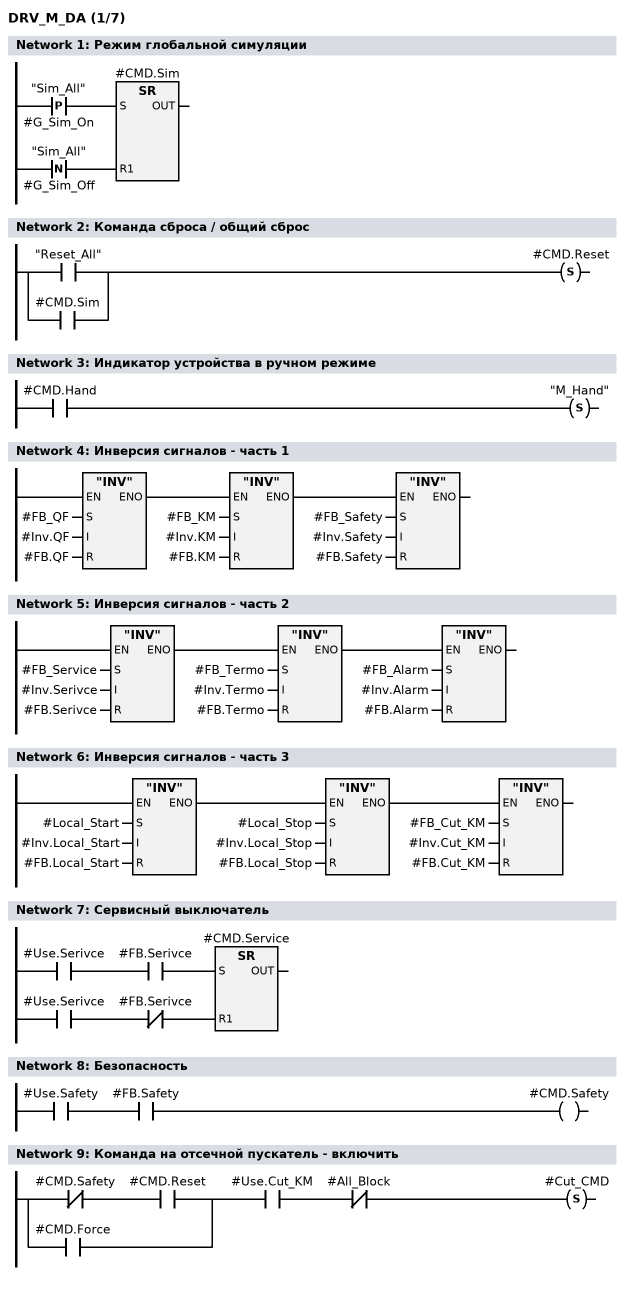
   RUNG wire#powerrail
      P_Contact(operand := "Sim_All", bit := #G_Sim_On)
      S_SR(operand := #CMD.Sim, r1 := wire#w1)
   END_RUNG
   RUNG wire#powerrail
      N_Contact(operand := "Sim_All", bit := #G_Sim_Off)
   END_RUNG wire#w1
   // the same network as SCL:
   #_w1 := "Sim_All" AND NOT #G_Sim_On;   // rising edge of "Sim_All"
   #G_Sim_On := "Sim_All";
   #_w2 := NOT "Sim_All" AND #G_Sim_Off;   // falling edge of "Sim_All"
   #G_Sim_Off := "Sim_All";
   IF #_w1 THEN
       #CMD.Sim := TRUE;   // SR flip-flop
   END_IF;
   IF #_w2 THEN #CMD.Sim := FALSE; END_IF;
END_REGION

REGION Network 2: Команда сброса / общий сброс
   RUNG wire#powerrail
      Contact( "Reset_All" )
      wire#w1
      S_Coil( #CMD.Reset )
   END_RUNG
   RUNG wire#powerrail
      Contact( #CMD.Sim )
   END_RUNG wire#w1
   // the same network as SCL:
   IF "Reset_All" OR #CMD.Sim THEN #CMD.Reset := TRUE; END_IF;
END_REGION

REGION Network 3: Индикатор устройства в ручном режиме
   RUNG wire#powerrail
      Contact( #CMD.Hand )
      S_Coil( "M_Hand" )
   END_RUNG
   // the same network as SCL:
   IF #CMD.Hand THEN "M_Hand" := TRUE; END_IF;
END_REGION

REGION Network 4: Инверсия сигналов - часть 1
   RUNG wire#powerrail
      "INV"(S := #FB_QF, I := #Inv.QF, R := #FB.QF)
      "INV"(S := #FB_KM, I := #Inv.KM, R := #FB.KM)
      "INV"(S := #FB_Safety, I := #Inv.Safety, R := #FB.Safety)
   END_RUNG
   // the same network as SCL:
   "INV"(S := #FB_QF, I := #Inv.QF, R := #FB.QF, ENO => #_w1);
   "INV"(EN := #_w1, S := #FB_KM, I := #Inv.KM, R := #FB.KM, ENO => #_w2);
   IF #_w2 THEN "INV"(S := #FB_Safety, I := #Inv.Safety, R := #FB.Safety); END_IF;
END_REGION

REGION Network 5: Инверсия сигналов - часть 2
   RUNG wire#powerrail
      "INV"(S := #FB_Service, I := #Inv.Serivce, R := #FB.Serivce)
      "INV"(S := #FB_Termo, I := #Inv.Termo, R := #FB.Termo)
      "INV"(S := #FB_Alarm, I := #Inv.Alarm, R := #FB.Alarm)
   END_RUNG
   // the same network as SCL:
   "INV"(S := #FB_Service, I := #Inv.Serivce, R := #FB.Serivce, ENO => #_w1);
   "INV"(EN := #_w1, S := #FB_Termo, I := #Inv.Termo, R := #FB.Termo, ENO => #_w2);
   IF #_w2 THEN "INV"(S := #FB_Alarm, I := #Inv.Alarm, R := #FB.Alarm); END_IF;
END_REGION

REGION Network 6: Инверсия сигналов - часть 3
   RUNG wire#powerrail
      "INV"(S := #Local_Start, I := #Inv.Local_Start, R := #FB.Local_Start)
      "INV"(S := #Local_Stop, I := #Inv.Local_Stop, R := #FB.Local_Stop)
      "INV"(S := #FB_Cut_KM, I := #Inv.Cut_KM, R := #FB.Cut_KM)
   END_RUNG
   // the same network as SCL:
   "INV"(S := #Local_Start, I := #Inv.Local_Start, R := #FB.Local_Start, ENO => #_w1);
   "INV"(EN := #_w1, S := #Local_Stop, I := #Inv.Local_Stop, R := #FB.Local_Stop, ENO => #_w2);
   IF #_w2 THEN "INV"(S := #FB_Cut_KM, I := #Inv.Cut_KM, R := #FB.Cut_KM); END_IF;
END_REGION

REGION Network 7: Сервисный выключатель
   RUNG wire#powerrail
      Contact( #Use.Serivce )
      Contact( #FB.Serivce )
      S_SR(operand := #CMD.Service, r1 := wire#w1)
   END_RUNG
   RUNG wire#powerrail
      Contact( #Use.Serivce )
      I_Contact( #FB.Serivce )
   END_RUNG wire#w1
   // the same network as SCL:
   IF #Use.Serivce AND #FB.Serivce THEN
       #CMD.Service := TRUE;   // SR flip-flop
   END_IF;
   IF #Use.Serivce AND NOT #FB.Serivce THEN #CMD.Service := FALSE; END_IF;
END_REGION

REGION Network 8: Безопасность
   RUNG wire#powerrail
      Contact( #Use.Safety )
      Contact( #FB.Safety )
      Coil( #CMD.Safety )
   END_RUNG
   // the same network as SCL:
   #CMD.Safety := #Use.Safety AND #FB.Safety;
END_REGION

REGION Network 9: Команда на отсечной пускатель - включить
   RUNG wire#powerrail
      I_Contact( #CMD.Safety )
      Contact( #CMD.Reset )
      wire#w1
      Contact( #Use.Cut_KM )
      I_Contact( #All_Block )
      S_Coil( #Cut_CMD )
   END_RUNG
   RUNG wire#powerrail
      Contact( #CMD.Force )
   END_RUNG wire#w1
   // the same network as SCL:
   IF ((NOT #CMD.Safety AND #CMD.Reset) OR #CMD.Force) AND #Use.Cut_KM AND NOT #All_Block THEN
       #Cut_CMD := TRUE;
   END_IF;
END_REGION

REGION Network 10: Команда на отсечной пускатель - выключить
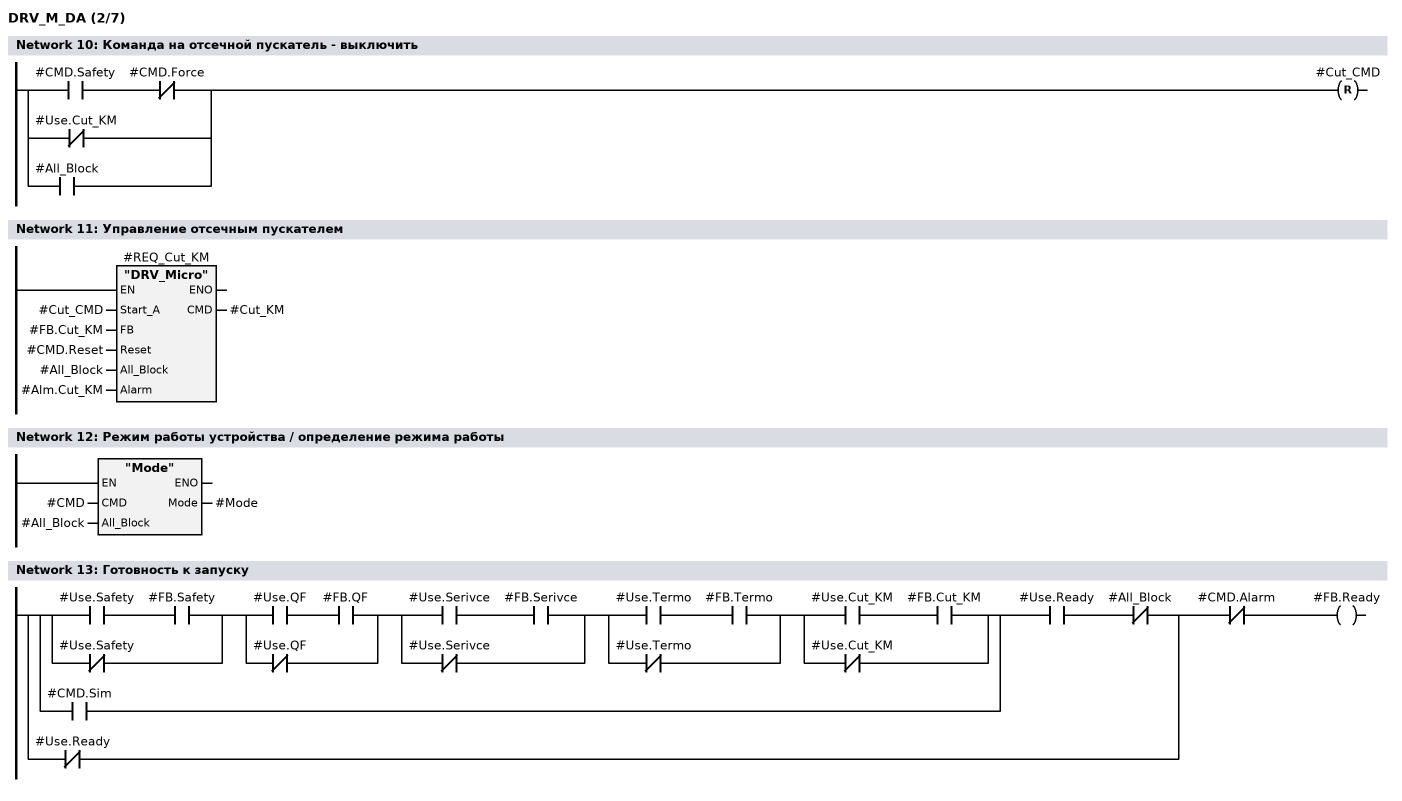
   RUNG wire#powerrail
      Contact( #CMD.Safety )
      I_Contact( #CMD.Force )
      wire#w1
      R_Coil( #Cut_CMD )
   END_RUNG
   RUNG wire#powerrail
      I_Contact( #Use.Cut_KM )
   END_RUNG wire#w1
   RUNG wire#powerrail
      Contact( #All_Block )
   END_RUNG wire#w1
   // the same network as SCL:
   IF (#CMD.Safety AND NOT #CMD.Force) OR NOT #Use.Cut_KM OR #All_Block THEN #Cut_CMD := FALSE; END_IF;
END_REGION

REGION Network 11: Управление отсечным пускателем
   RUNG wire#powerrail
      #REQ_Cut_KM(Start_A := #Cut_CMD, FB := #FB.Cut_KM, Reset := #CMD.Reset, All_Block := #All_Block, Alarm := #Alm.Cut_KM, CMD => #Cut_KM)
   END_RUNG
   // the same network as SCL:
   #REQ_Cut_KM(Start_A := #Cut_CMD,   // "DRV_Micro"
               FB := #FB.Cut_KM,
               Reset := #CMD.Reset,
               All_Block := #All_Block,
               Alarm := #Alm.Cut_KM,
               CMD => #Cut_KM);
END_REGION

REGION Network 12: Режим работы устройства / определение режима работы
   RUNG wire#powerrail
      "Mode"(CMD := #CMD, All_Block := #All_Block, Mode => #Mode)
   END_RUNG
   // the same network as SCL:
   "Mode"(CMD := #CMD, All_Block := #All_Block, Mode => #Mode);
END_REGION

REGION Network 13: Готовность к запуску
   RUNG wire#powerrail
      Contact( #Use.Safety )
      Contact( #FB.Safety )
      wire#w1
      Contact( #Use.QF )
      Contact( #FB.QF )
      wire#w2
      Contact( #Use.Serivce )
      Contact( #FB.Serivce )
      wire#w3
      Contact( #Use.Termo )
      Contact( #FB.Termo )
      wire#w4
      Contact( #Use.Cut_KM )
      Contact( #FB.Cut_KM )
      wire#w5
      Contact( #Use.Ready )
      I_Contact( #All_Block )
      wire#w6
      I_Contact( #CMD.Alarm )
      Coil( #FB.Ready )
   END_RUNG
   RUNG wire#powerrail
      I_Contact( #Use.Safety )
   END_RUNG wire#w1
   RUNG wire#w1
      I_Contact( #Use.QF )
   END_RUNG wire#w2
   RUNG wire#w2
      I_Contact( #Use.Serivce )
   END_RUNG wire#w3
   RUNG wire#w3
      I_Contact( #Use.Termo )
   END_RUNG wire#w4
   RUNG wire#w4
      I_Contact( #Use.Cut_KM )
   END_RUNG wire#w5
   RUNG wire#powerrail
      Contact( #CMD.Sim )
   END_RUNG wire#w5
   RUNG wire#powerrail
      I_Contact( #Use.Ready )
   END_RUNG wire#w6
   // the same network as SCL:
   #FB.Ready := ((((((#Use.Safety AND #FB.Safety) OR NOT #Use.Safety) AND ((#Use.QF AND #FB.QF) OR NOT #Use.QF) AND ((#Use.Serivce AND #FB.Serivce) OR NOT #Use.Serivce) AND ((#Use.Termo AND #FB.Termo) OR NOT #Use.Termo) AND ((#Use.Cut_KM AND #FB.Cut_KM) OR NOT #Use.Cut_KM)) OR #CMD.Sim) AND #Use.Ready AND NOT #All_Block) OR NOT #Use.Ready) AND NOT #CMD.Alarm;
END_REGION

REGION Network 14: Управление запуском / дискретный управляющий сигнал
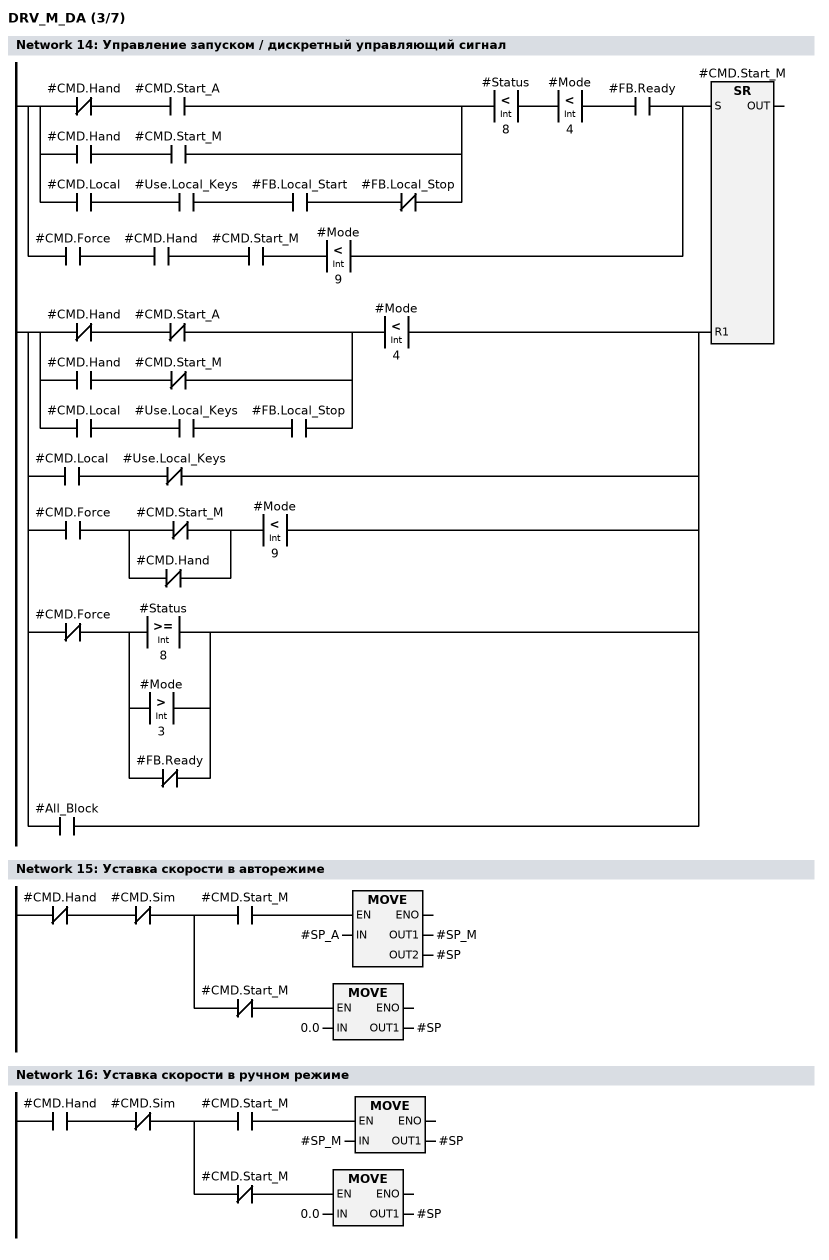
   RUNG wire#powerrail
      I_Contact( #CMD.Hand )
      Contact( #CMD.Start_A )
      wire#w1
      { S7_Templates := "SrcType := Int" } LT_Contact(in1 := #Status, in2 := 8)
      { S7_Templates := "SrcType := Int" } LT_Contact(in1 := #Mode, in2 := 4)
      Contact( #FB.Ready )
      wire#w2
      S_SR(operand := #CMD.Start_M, r1 := wire#w7)
   END_RUNG
   RUNG wire#powerrail
      Contact( #CMD.Hand )
      Contact( #CMD.Start_M )
   END_RUNG wire#w1
   RUNG wire#powerrail
      Contact( #CMD.Local )
      Contact( #Use.Local_Keys )
      Contact( #FB.Local_Start )
      I_Contact( #FB.Local_Stop )
   END_RUNG wire#w1
   RUNG wire#powerrail
      Contact( #CMD.Force )
      Contact( #CMD.Hand )
      Contact( #CMD.Start_M )
      { S7_Templates := "SrcType := Int" } LT_Contact(in1 := #Mode, in2 := 9)
   END_RUNG wire#w2
   RUNG wire#powerrail
      I_Contact( #CMD.Hand )
      I_Contact( #CMD.Start_A )
      wire#w3
      { S7_Templates := "SrcType := Int" } LT_Contact(in1 := #Mode, in2 := 4)
   END_RUNG wire#w7
   RUNG wire#powerrail
      Contact( #CMD.Hand )
      I_Contact( #CMD.Start_M )
   END_RUNG wire#w3
   RUNG wire#powerrail
      Contact( #CMD.Local )
      Contact( #Use.Local_Keys )
      Contact( #FB.Local_Stop )
   END_RUNG wire#w3
   RUNG wire#powerrail
      Contact( #CMD.Local )
      I_Contact( #Use.Local_Keys )
   END_RUNG wire#w7
   RUNG wire#powerrail
      Contact( #CMD.Force )
      wire#w4
      I_Contact( #CMD.Start_M )
      wire#w5
      { S7_Templates := "SrcType := Int" } LT_Contact(in1 := #Mode, in2 := 9)
   END_RUNG wire#w7
   RUNG wire#w4
      I_Contact( #CMD.Hand )
   END_RUNG wire#w5
   RUNG wire#powerrail
      I_Contact( #CMD.Force )
      wire#w6
      { S7_Templates := "SrcType := Int" } GE_Contact(in1 := #Status, in2 := 8)
   END_RUNG wire#w7
   RUNG wire#w6
      { S7_Templates := "SrcType := Int" } GT_Contact(in1 := #Mode, in2 := 3)
   END_RUNG wire#w7
   RUNG wire#w6
      I_Contact( #FB.Ready )
   END_RUNG wire#w7
   RUNG wire#powerrail
      Contact( #All_Block )
   END_RUNG wire#w7
   // the same network as SCL:
   #_w1 := (((NOT #CMD.Hand AND NOT #CMD.Start_A) OR (#CMD.Hand AND NOT #CMD.Start_M) OR (#CMD.Local AND #Use.Local_Keys AND #FB.Local_Stop)) AND (#Mode < 4)) OR (#CMD.Local AND NOT #Use.Local_Keys) OR (#CMD.Force AND (NOT #CMD.Start_M OR NOT #CMD.Hand) AND (#Mode < 9)) OR (NOT #CMD.Force AND ((#Status >= 8) OR (#Mode > 3) OR NOT #FB.Ready)) OR #All_Block;
   IF (((NOT #CMD.Hand AND #CMD.Start_A) OR (#CMD.Hand AND #CMD.Start_M) OR (#CMD.Local AND #Use.Local_Keys AND #FB.Local_Start AND NOT #FB.Local_Stop)) AND (#Status < 8) AND (#Mode < 4) AND #FB.Ready) OR (#CMD.Force AND #CMD.Hand AND #CMD.Start_M AND (#Mode < 9)) THEN
       #CMD.Start_M := TRUE;   // SR flip-flop
   END_IF;
   IF #_w1 THEN #CMD.Start_M := FALSE; END_IF;
END_REGION

REGION Network 15: Уставка скорости в авторежиме
   RUNG wire#powerrail
      I_Contact( #CMD.Hand )
      I_Contact( #CMD.Sim )
      wire#w1
      Contact( #CMD.Start_M )
      Move(in := #SP_A, out1 => #SP_M, out2 => #SP)
   END_RUNG
   RUNG wire#w1
      I_Contact( #CMD.Start_M )
      Move(in := 0.0, out1 => #SP)
   END_RUNG
   // the same network as SCL:
   #_w1 := NOT #CMD.Hand AND NOT #CMD.Sim;
   IF #_w1 AND #CMD.Start_M THEN
       #SP_M := #SP_A;
       #SP := #SP_A;
   END_IF;
   IF #_w1 AND NOT #CMD.Start_M THEN #SP := 0.0; END_IF;
END_REGION

REGION Network 16: Уставка скорости в ручном режиме
   RUNG wire#powerrail
      Contact( #CMD.Hand )
      I_Contact( #CMD.Sim )
      wire#w1
      Contact( #CMD.Start_M )
      Move(in := #SP_M, out1 => #SP)
   END_RUNG
   RUNG wire#w1
      I_Contact( #CMD.Start_M )
      Move(in := 0.0, out1 => #SP)
   END_RUNG
   // the same network as SCL:
   #_w1 := #CMD.Hand AND NOT #CMD.Sim;
   IF #_w1 AND #CMD.Start_M THEN #SP := #SP_M; END_IF;
   IF #_w1 AND NOT #CMD.Start_M THEN #SP := 0.0; END_IF;
END_REGION

REGION Network 17: Задержка пуска
